LIN {X -0.068,Y -157.540,Z 1544.848,A 0.000,B 0.000,C 90.000,E1 152.615} C_DIS
LIN {X 0.098,Y -161.777,Z 1544.828,A 0.000,B 0.000,C 90.000,E1 148.997} C_DIS
LIN {X -0.019,Y -165.970,Z 1544.808,A 0.000,B 0.000,C 90.000,E1 145.515} C_DIS
LIN {X -0.024,Y -170.964,Z 1544.789,A 0.000,B 0.000,C 90.000,E1 142.029} C_DIS
LIN {X 0.028,Y -175.833,Z 1544.770,A 0.000,B 0.000,C 90.000,E1 138.566} C_DIS
LIN {X 0.023,Y -181.439,Z 1544.751,A 0.000,B 0.000,C 90.000,E1 135.162} C_DIS
LIN {X -0.103,Y -186.945,Z 1544.732,A 0.000,B 0.000,C 90.000,E1 131.838} C_DIS
LIN {X -0.104,Y -190.058,Z 1544.723,A 0.000,B 0.000,C 90.000,E1 130.172} C_DIS
LIN {X -0.090,Y -195.833,Z 1544.705,A 0.000,B 0.000,C 90.000,E1 126.870} C_DIS
LIN {X -0.023,Y -200.665,Z 1544.691,A 0.000,B 0.000,C 90.000,E1 124.405} C_DIS
LIN {X -0.041,Y -203.117,Z 1544.683,A 0.000,B 0.000,C 90.000,E1 123.007} C_DIS
LIN {X 0.168,Y -318.490,Z 1544.683,A 0.000,B 0.000,C 90.000,E1 122.959} C_DIS
LIN {X 0.099,Y -319.542,Z 1544.683,A 0.000,B 0.000,C 90.000,E1 122.959} C_DIS
LIN {X 0.174,Y -324.477,Z 1544.682,A 0.000,B 0.000,C 90.000,E1 122.752} C_DIS
LIN {X -0.044,Y -327.554,Z 1544.681,A 0.000,B 0.000,C 90.000,E1 122.546} C_DIS
LIN {X -0.058,Y -331.261,Z 1544.678,A 0.000,B 0.000,C 90.000,E1 122.084} C_DIS
LIN {X 0.052,Y -333.020,Z 1544.676,A 0.000,B 0.000,C 90.000,E1 121.750} C_DIS
LIN {X 0.134,Y -336.789,Z 1544.671,A 0.000,B 0.000,C 90.000,E1 120.797} C_DIS
LIN {X 0.103,Y -348.404,Z 1544.656,A 0.000,B 0.000,C 90.000,E1 118.025} C_DIS
LIN {X -0.101,Y -361.451,Z 1544.641,A 0.000,B 0.000,C 90.000,E1 115.335} C_DIS
LIN {X 0.095,Y -376.031,Z 1544.626,A 0.000,B 0.000,C 90.000,E1 112.642} C_DIS
LIN {X -0.090,Y -390.387,Z 1544.613,A 0.000,B 0.000,C 90.000,E1 110.355} C_DIS
LIN {X 0.177,Y -406.158,Z 1544.600,A 0.000,B 0.000,C 90.000,E1 108.055} C_DIS
LIN {X 0.216,Y -423.455,Z 1544.588,A 0.000,B 0.000,C 90.000,E1 105.843} C_DIS
LIN {X 0.058,Y -442.382,Z 1544.576,A 0.000,B 0.000,C 90.000,E1 103.716} C_DIS
LIN {X -0.096,Y -462.375,Z 1544.565,A 0.000,B 0.000,C 90.000,E1 101.715} C_DIS
LIN {X 0.079,Y -485.531,Z 1544.553,A 0.000,B 0.000,C 90.000,E1 99.613} C_DIS
LIN {X 0.000,Y -493.167,Z 1544.550,A 0.000,B 0.000,C 90.000,E1 98.973} C_DIS
LIN {X 0.111,Y -494.997,Z 1544.549,A 0.000,B 0.000,C 90.000,E1 98.746} C_DIS
LIN {X 0.025,Y -496.592,Z 1544.547,A 0.000,B 0.000,C 90.000,E1 98.511} C_DIS
LIN {X -0.065,Y -497.782,Z 1544.546,A 0.000,B 0.000,C 90.000,E1 98.276} C_DIS
LIN {X 0.196,Y -499.207,Z 1544.543,A 0.000,B 0.000,C 90.000,E1 97.757} C_DIS
LIN {X -0.028,Y -499.572,Z 1544.541,A 0.000,B 0.000,C 90.000,E1 97.296} C_DIS
LIN {X -0.244,Y -498.940,Z 1544.538,A 0.000,B 0.000,C 90.000,E1 96.834} C_DIS
LIN {X 0.037,Y -497.207,Z 1544.535,A 0.000,B 0.000,C 90.000,E1 96.315} C_DIS
LIN {X -0.097,Y -495.828,Z 1544.534,A 0.000,B 0.000,C 90.000,E1 96.087} C_DIS
LIN {X -0.001,Y -484.503,Z 1544.524,A 0.000,B 0.000,C 90.000,E1 94.359} C_DIS
LIN {X 0.011,Y -475.130,Z 1544.516,A 0.000,B 0.000,C 90.000,E1 92.865} C_DIS
LIN {X 0.033,Y -466.858,Z 1544.509,A 0.000,B 0.000,C 90.000,E1 91.604} C_DIS
LIN {X 0.171,Y -456.481,Z 1544.500,A 0.000,B 0.000,C 90.000,E1 90.057} C_DIS
LIN {X -0.075,Y -447.464,Z 1544.493,A 0.000,B 0.000,C 90.000,E1 88.797} C_DIS
LIN {X 0.005,Y -438.078,Z 1544.486,A 0.000,B 0.000,C 90.000,E1 87.478} C_DIS
LIN {X 0.117,Y -426.571,Z 1544.477,A 0.000,B 0.000,C 90.000,E1 85.869} C_DIS
LIN {X 0.117,Y -413.092,Z 1544.467,A 0.000,B 0.000,C 90.000,E1 83.976} C_DIS
LIN {X 0.005,Y -398.136,Z 1544.454,A 0.000,B 0.000,C 90.000,E1 81.781} C_DIS
LIN {X 0.140,Y -380.438,Z 1544.439,A 0.000,B 0.000,C 90.000,E1 78.926} C_DIS
LIN {X -0.080,Y -363.765,Z 1544.422,A 0.000,B 0.000,C 90.000,E1 76.047} C_DIS
LIN {X 0.113,Y -350.852,Z 1544.409,A 0.000,B 0.000,C 90.000,E1 73.630} C_DIS
LIN {X 0.038,Y -341.231,Z 1544.399,A 0.000,B 0.000,C 90.000,E1 71.819} C_DIS
LIN {X 0.006,Y -325.755,Z 1544.382,A 0.000,B 0.000,C 90.000,E1 68.720} C_DIS
LIN {X -0.096,Y -309.683,Z 1544.362,A 0.000,B 0.000,C 90.000,E1 65.229} C_DIS
LIN {X 0.022,Y -299.787,Z 1544.350,A 0.000,B 0.000,C 90.000,E1 62.922} C_DIS
LIN {X 0.049,Y -288.590,Z 1544.335,A 0.000,B 0.000,C 90.000,E1 60.255} C_DIS
LIN {X -0.083,Y -280.298,Z 1544.323,A 0.000,B 0.000,C 90.000,E1 58.250} C_DIS
LIN {X 0.030,Y -269.427,Z 1544.308,A 0.000,B 0.000,C 90.000,E1 55.468} C_DIS
LIN {X 0.095,Y -258.999,Z 1544.293,A 0.000,B 0.000,C 90.000,E1 52.637} C_DIS
LIN {X -0.168,Y -247.742,Z 1544.275,A 0.000,B 0.000,C 90.000,E1 49.461} C_DIS
LIN {X -0.080,Y -237.298,Z 1544.256,A 0.000,B 0.000,C 90.000,E1 46.134} C_DIS
LIN {X -0.066,Y -228.747,Z 1544.240,A 0.000,B 0.000,C 90.000,E1 43.137} C_DIS
LIN {X -0.059,Y -221.025,Z 1544.223,A 0.000,B 0.000,C 90.000,E1 40.092} C_DIS
LIN {X -0.046,Y -214.000,Z 1544.205,A 0.000,B 0.000,C 90.000,E1 36.996} C_DIS
LIN {X 0.043,Y -207.763,Z 1544.188,A 0.000,B 0.000,C 90.000,E1 33.833} C_DIS
LIN {X -0.017,Y -202.302,Z 1544.170,A 0.000,B 0.000,C 90.000,E1 30.669} C_DIS
LIN {X -0.055,Y -197.586,Z 1544.152,A 0.000,B 0.000,C 90.000,E1 27.462} C_DIS
LIN {X -0.029,Y -192.589,Z 1544.130,A 0.000,B 0.000,C 90.000,E1 23.387} C_DIS
LIN {X -0.010,Y -188.278,Z 1544.107,A 0.000,B 0.000,C 90.000,E1 19.268} C_DIS
LIN {X -0.067,Y -184.100,Z 1544.079,A 0.000,B 0.000,C 90.000,E1 14.300} C_DIS
LIN {X -0.049,Y -180.889,Z 1544.051,A 0.000,B 0.000,C 90.000,E1 9.265} C_DIS
LIN {X 0.079,Y -178.282,Z 1544.014,A 0.000,B 0.000,C 90.000,E1 2.465} C_DIS
LIN {X -0.010,Y -178.518,Z 1543.955,A 0.000,B 0.000,C 90.000,E1 351.894} C_DIS
LIN {X 0.095,Y -180.978,Z 1543.922,A 0.000,B 0.000,C 90.000,E1 345.936} C_DIS
LIN {X 0.017,Y -184.467,Z 1543.894,A 0.000,B 0.000,C 90.000,E1 340.913} C_DIS
LIN {X 0.011,Y -188.390,Z 1543.871,A 0.000,B 0.000,C 90.000,E1 336.741} C_DIS
LIN {X -0.016,Y -193.357,Z 1543.848,A 0.000,B 0.000,C 90.000,E1 332.615} C_DIS
LIN {X -0.043,Y -199.165,Z 1543.825,A 0.000,B 0.000,C 90.000,E1 328.535} C_DIS
LIN {X -0.061,Y -204.509,Z 1543.807,A 0.000,B 0.000,C 90.000,E1 325.308} C_DIS
LIN {X -0.042,Y -210.670,Z 1543.789,A 0.000,B 0.000,C 90.000,E1 322.110} C_DIS
LIN {X 0.060,Y -217.651,Z 1543.772,A 0.000,B 0.000,C 90.000,E1 318.933} C_DIS
LIN {X -0.094,Y -226.415,Z 1543.753,A 0.000,B 0.000,C 90.000,E1 315.486} C_DIS
LIN {X 0.019,Y -236.333,Z 1543.734,A 0.000,B 0.000,C 90.000,E1 312.043} C_DIS
LIN {X 0.035,Y -242.594,Z 1543.723,A 0.000,B 0.000,C 90.000,E1 310.172} C_DIS
LIN {X 0.000,Y -248.230,Z 1543.715,A 0.000,B 0.000,C 90.000,E1 308.705} C_DIS
LIN {X 0.053,Y -256.174,Z 1543.705,A 0.000,B 0.000,C 90.000,E1 306.870} C_DIS
LIN {X -0.071,Y -265.290,Z 1543.695,A 0.000,B 0.000,C 90.000,E1 305.105} C_DIS
LIN {X 0.166,Y -275.499,Z 1543.685,A 0.000,B 0.000,C 90.000,E1 303.293} C_DIS
LIN {X -0.023,Y -291.443,Z 1543.672,A 0.000,B 0.000,C 90.000,E1 300.924} C_DIS
LIN {X 0.132,Y -311.376,Z 1543.657,A 0.000,B 0.000,C 90.000,E1 298.231} C_DIS
LIN {X -0.178,Y -326.813,Z 1543.646,A 0.000,B 0.000,C 90.000,E1 296.360} C_DIS
LIN {X 0.031,Y -345.069,Z 1543.634,A 0.000,B 0.000,C 90.000,E1 294.155} C_DIS
LIN {X 0.097,Y -363.451,Z 1543.623,A 0.000,B 0.000,C 90.000,E1 292.099} C_DIS
LIN {X -0.075,Y -376.354,Z 1543.615,A 0.000,B 0.000,C 90.000,E1 290.737} C_DIS
LIN {X 0.093,Y -386.609,Z 1543.609,A 0.000,B 0.000,C 90.000,E1 289.577} C_DIS
LIN {X 0.042,Y -393.934,Z 1543.604,A 0.000,B 0.000,C 90.000,E1 288.725} C_DIS
LIN {X 0.046,Y -400.651,Z 1543.599,A 0.000,B 0.000,C 90.000,E1 287.873} C_DIS
LIN {X -0.003,Y -406.701,Z 1543.595,A 0.000,B 0.000,C 90.000,E1 287.040} C_DIS
LIN {X 0.000,Y -412.021,Z 1543.590,A 0.000,B 0.000,C 90.000,E1 286.205} C_DIS
LIN {X -0.064,Y -415.120,Z 1543.587,A 0.000,B 0.000,C 90.000,E1 285.662} C_DIS
LIN {X 0.020,Y -419.032,Z 1543.582,A 0.000,B 0.000,C 90.000,E1 284.828} C_DIS
LIN {X 0.032,Y -422.199,Z 1543.578,A 0.000,B 0.000,C 90.000,E1 284.008} C_DIS
LIN {X -0.083,Y -423.934,Z 1543.575,A 0.000,B 0.000,C 90.000,E1 283.480} C_DIS
LIN {X -0.089,Y -425.263,Z 1543.572,A 0.000,B 0.000,C 90.000,E1 282.939} C_DIS
LIN {X 0.233,Y -426.168,Z 1543.569,A 0.000,B 0.000,C 90.000,E1 282.355} C_DIS
LIN {X 0.147,Y -426.651,Z 1543.566,A 0.000,B 0.000,C 90.000,E1 281.827} C_DIS
LIN {X 0.065,Y -426.619,Z 1543.563,A 0.000,B 0.000,C 90.000,E1 281.299} C_DIS
LIN {X -0.095,Y -426.088,Z 1543.560,A 0.000,B 0.000,C 90.000,E1 280.782} C_DIS
LIN {X -0.173,Y -424.963,Z 1543.557,A 0.000,B 0.000,C 90.000,E1 280.254} C_DIS
LIN {X 0.160,Y -423.171,Z 1543.554,A 0.000,B 0.000,C 90.000,E1 279.670} C_DIS
LIN {X -0.001,Y -420.757,Z 1543.551,A 0.000,B 0.000,C 90.000,E1 279.151} C_DIS
LIN {X -0.111,Y -417.535,Z 1543.548,A 0.000,B 0.000,C 90.000,E1 278.624} C_DIS
LIN {X 0.111,Y -413.410,Z 1543.545,A 0.000,B 0.000,C 90.000,E1 278.049} C_DIS
LIN {X -0.094,Y -408.430,Z 1543.542,A 0.000,B 0.000,C 90.000,E1 277.530} C_DIS
LIN {X -0.168,Y -402.630,Z 1543.539,A 0.000,B 0.000,C 90.000,E1 277.004} C_DIS
LIN {X 0.090,Y -396.635,Z 1543.536,A 0.000,B 0.000,C 90.000,E1 276.486} C_DIS
LIN {X -0.193,Y -390.365,Z 1543.534,A 0.000,B 0.000,C 90.000,E1 276.087} C_DIS
LIN {X -0.094,Y -384.023,Z 1543.531,A 0.000,B 0.000,C 90.000,E1 275.682} C_DIS
LIN {X -0.026,Y -374.466,Z 1543.529,A 0.000,B 0.000,C 90.000,E1 275.163} C_DIS
LIN {X 0.057,Y -364.853,Z 1543.526,A 0.000,B 0.000,C 90.000,E1 274.702} C_DIS
LIN {X -0.156,Y -352.144,Z 1543.523,A 0.000,B 0.000,C 90.000,E1 274.188} C_DIS
LIN {X -0.069,Y -342.518,Z 1543.521,A 0.000,B 0.000,C 90.000,E1 273.784} C_DIS
LIN {X 0.158,Y -332.329,Z 1543.519,A 0.000,B 0.000,C 90.000,E1 273.383} C_DIS
LIN {X 0.116,Y -319.217,Z 1543.517,A 0.000,B 0.000,C 90.000,E1 272.980} C_DIS
LIN {X -0.130,Y -309.122,Z 1543.515,A 0.000,B 0.000,C 90.000,E1 272.751} C_DIS
LIN {X 0.095,Y -297.890,Z 1543.514,A 0.000,B 0.000,C 90.000,E1 272.465} C_DIS
LIN {X -0.025,Y -285.540,Z 1543.513,A 0.000,B 0.000,C 90.000,E1 272.293} C_DIS
LIN {X -0.121,Y -272.247,Z 1543.512,A 0.000,B 0.000,C 90.000,E1 272.178} C_DIS
LIN {X 0.101,Y -260.337,Z 1543.512,A 0.000,B 0.000,C 90.000,E1 272.064} C_DIS
LIN {X 0.037,Y -181.250,Z 1543.511,A 0.000,B 0.000,C 90.000,E1 272.064} C_DIS
LIN {X 0.052,Y -181.579,Z 1543.502,A 0.000,B 0.000,C 90.000,E1 270.344} C_DIS
LIN {X 0.027,Y -180.905,Z 1543.474,A 0.000,B 0.000,C 90.000,E1 265.298} C_DIS
LIN {X -0.023,Y -180.248,Z 1543.465,A 0.000,B 0.000,C 90.000,E1 263.628} C_DIS
LIN {X -0.004,Y -178.736,Z 1543.441,A 0.000,B 0.000,C 90.000,E1 259.398} C_DIS
LIN {X 0.063,Y -175.783,Z 1543.413,A 0.000,B 0.000,C 90.000,E1 254.283} C_DIS
LIN {X 0.051,Y -171.968,Z 1543.384,A 0.000,B 0.000,C 90.000,E1 249.156} C_DIS
LIN {X 0.088,Y -171.367,Z 1543.380,A 0.000,B 0.000,C 90.000,E1 248.284} C_DIS
LIN {X -0.085,Y -167.614,Z 1543.355,A 0.000,B 0.000,C 90.000,E1 244.024} C_DIS
LIN {X 0.077,Y -166.264,Z 1543.346,A 0.000,B 0.000,C 90.000,E1 242.231} C_DIS
LIN {X 0.064,Y -163.016,Z 1543.326,A 0.000,B 0.000,C 90.000,E1 238.742} C_DIS
LIN {X -0.023,Y -160.941,Z 1543.312,A 0.000,B 0.000,C 90.000,E1 236.135} C_DIS
LIN {X 0.087,Y -157.699,Z 1543.292,A 0.000,B 0.000,C 90.000,E1 232.557} C_DIS
LIN {X 0.025,Y -155.738,Z 1543.277,A 0.000,B 0.000,C 90.000,E1 229.908} C_DIS
LIN {X 0.078,Y -151.996,Z 1543.252,A 0.000,B 0.000,C 90.000,E1 225.405} C_DIS
LIN {X 0.094,Y -150.241,Z 1543.237,A 0.000,B 0.000,C 90.000,E1 222.690} C_DIS
LIN {X 0.017,Y -147.000,Z 1543.212,A 0.000,B 0.000,C 90.000,E1 218.177} C_DIS
LIN {X 0.006,Y -145.585,Z 1543.197,A 0.000,B 0.000,C 90.000,E1 215.438} C_DIS
LIN {X 0.000,Y -142.973,Z 1543.171,A 0.000,B 0.000,C 90.000,E1 210.846} C_DIS
LIN {X 0.054,Y -141.600,Z 1543.151,A 0.000,B 0.000,C 90.000,E1 207.129} C_DIS
LIN {X -0.031,Y -139.423,Z 1543.115,A 0.000,B 0.000,C 90.000,E1 200.663} C_DIS
LIN {X 0.020,Y -139.151,Z 1543.104,A 0.000,B 0.000,C 90.000,E1 198.779} C_DIS
LIN {X 0.043,Y -138.345,Z 1543.058,A 0.000,B 0.000,C 90.000,E1 190.366} C_DIS
LIN {X 0.028,Y -139.485,Z 1543.006,A 0.000,B 0.000,C 90.000,E1 181.031} C_DIS
LIN {X -0.032,Y -141.084,Z 1542.975,A 0.000,B 0.000,C 90.000,E1 175.469} C_DIS
LIN {X 0.062,Y -142.461,Z 1542.959,A 0.000,B 0.000,C 90.000,E1 172.648} C_DIS
LIN {X 0.011,Y -144.706,Z 1542.934,A 0.000,B 0.000,C 90.000,E1 168.049} C_DIS
LIN {X -0.037,Y -147.303,Z 1542.913,A 0.000,B 0.000,C 90.000,E1 164.393} C_DIS
LIN {X -0.022,Y -150.623,Z 1542.888,A 0.000,B 0.000,C 90.000,E1 159.826} C_DIS
LIN {X 0.055,Y -154.098,Z 1542.868,A 0.000,B 0.000,C 90.000,E1 156.177} C_DIS
LIN {X -0.022,Y -157.521,Z 1542.848,A 0.000,B 0.000,C 90.000,E1 152.615} C_DIS
LIN {X -0.077,Y -161.755,Z 1542.828,A 0.000,B 0.000,C 90.000,E1 149.076} C_DIS
LIN {X 0.029,Y -165.948,Z 1542.808,A 0.000,B 0.000,C 90.000,E1 145.515} C_DIS
LIN {X 0.026,Y -170.939,Z 1542.789,A 0.000,B 0.000,C 90.000,E1 142.029} C_DIS
LIN {X -0.054,Y -175.807,Z 1542.770,A 0.000,B 0.000,C 90.000,E1 138.609} C_DIS
LIN {X 0.074,Y -181.415,Z 1542.751,A 0.000,B 0.000,C 90.000,E1 135.162} C_DIS
LIN {X -0.052,Y -186.918,Z 1542.732,A 0.000,B 0.000,C 90.000,E1 131.838} C_DIS
LIN {X 0.022,Y -191.496,Z 1542.719,A 0.000,B 0.000,C 90.000,E1 129.322} C_DIS
LIN {X 0.106,Y -197.359,Z 1542.700,A 0.000,B 0.000,C 90.000,E1 126.011} C_DIS
LIN {X 0.032,Y -200.636,Z 1542.691,A 0.000,B 0.000,C 90.000,E1 124.405} C_DIS
LIN {X -0.025,Y -203.053,Z 1542.683,A 0.000,B 0.000,C 90.000,E1 123.038} C_DIS
LIN {X -0.077,Y -318.319,Z 1542.683,A 0.000,B 0.000,C 90.000,E1 123.038} C_DIS
LIN {X -0.012,Y -324.630,Z 1542.682,A 0.000,B 0.000,C 90.000,E1 122.801} C_DIS
LIN {X 0.056,Y -327.580,Z 1542.681,A 0.000,B 0.000,C 90.000,E1 122.546} C_DIS
LIN {X -0.033,Y -331.300,Z 1542.678,A 0.000,B 0.000,C 90.000,E1 122.084} C_DIS
LIN {X 0.077,Y -333.015,Z 1542.677,A 0.000,B 0.000,C 90.000,E1 121.750} C_DIS
LIN {X -0.029,Y -339.215,Z 1542.668,A 0.000,B 0.000,C 90.000,E1 120.207} C_DIS
LIN {X 0.003,Y -351.135,Z 1542.652,A 0.000,B 0.000,C 90.000,E1 117.436} C_DIS
LIN {X 0.044,Y -364.510,Z 1542.637,A 0.000,B 0.000,C 90.000,E1 114.719} C_DIS
LIN {X -0.009,Y -379.447,Z 1542.623,A 0.000,B 0.000,C 90.000,E1 112.078} C_DIS
LIN {X 0.114,Y -394.145,Z 1542.610,A 0.000,B 0.000,C 90.000,E1 109.758} C_DIS
LIN {X 0.105,Y -410.284,Z 1542.597,A 0.000,B 0.000,C 90.000,E1 107.511} C_DIS
LIN {X 0.128,Y -427.977,Z 1542.585,A 0.000,B 0.000,C 90.000,E1 105.315} C_DIS
LIN {X 0.237,Y -447.270,Z 1542.573,A 0.000,B 0.000,C 90.000,E1 103.175} C_DIS
LIN {X -0.135,Y -467.405,Z 1542.562,A 0.000,B 0.000,C 90.000,E1 101.243} C_DIS
LIN {X -0.167,Y -490.700,Z 1542.551,A 0.000,B 0.000,C 90.000,E1 99.208} C_DIS
LIN {X 0.018,Y -493.100,Z 1542.550,A 0.000,B 0.000,C 90.000,E1 98.973} C_DIS
LIN {X 0.129,Y -494.921,Z 1542.549,A 0.000,B 0.000,C 90.000,E1 98.746} C_DIS
LIN {X 0.042,Y -496.509,Z 1542.547,A 0.000,B 0.000,C 90.000,E1 98.511} C_DIS
LIN {X -0.047,Y -497.693,Z 1542.546,A 0.000,B 0.000,C 90.000,E1 98.276} C_DIS
LIN {X 0.214,Y -499.108,Z 1542.543,A 0.000,B 0.000,C 90.000,E1 97.757} C_DIS
LIN {X -0.011,Y -499.466,Z 1542.541,A 0.000,B 0.000,C 90.000,E1 97.296} C_DIS
LIN {X -0.228,Y -498.826,Z 1542.538,A 0.000,B 0.000,C 90.000,E1 96.834} C_DIS
LIN {X 0.053,Y -497.084,Z 1542.535,A 0.000,B 0.000,C 90.000,E1 96.315} C_DIS
LIN {X -0.083,Y -495.699,Z 1542.534,A 0.000,B 0.000,C 90.000,E1 96.087} C_DIS
LIN {X 0.011,Y -484.387,Z 1542.524,A 0.000,B 0.000,C 90.000,E1 94.359} C_DIS
LIN {X 0.021,Y -475.033,Z 1542.516,A 0.000,B 0.000,C 90.000,E1 92.865} C_DIS
LIN {X 0.042,Y -466.753,Z 1542.509,A 0.000,B 0.000,C 90.000,E1 91.604} C_DIS
LIN {X -0.060,Y -458.152,Z 1542.502,A 0.000,B 0.000,C 90.000,E1 90.344} C_DIS
LIN {X 0.167,Y -449.206,Z 1542.495,A 0.000,B 0.000,C 90.000,E1 89.026} C_DIS
LIN {X 0.009,Y -438.010,Z 1542.486,A 0.000,B 0.000,C 90.000,E1 87.478} C_DIS
LIN {X -0.044,Y -428.469,Z 1542.479,A 0.000,B 0.000,C 90.000,E1 86.159} C_DIS
LIN {X 0.118,Y -413.097,Z 1542.467,A 0.000,B 0.000,C 90.000,E1 83.976} C_DIS
LIN {X 0.007,Y -398.158,Z 1542.454,A 0.000,B 0.000,C 90.000,E1 81.781} C_DIS
LIN {X 0.169,Y -378.752,Z 1542.437,A 0.000,B 0.000,C 90.000,E1 78.634} C_DIS
LIN {X -0.128,Y -360.518,Z 1542.419,A 0.000,B 0.000,C 90.000,E1 75.463} C_DIS
LIN {X 0.074,Y -347.664,Z 1542.406,A 0.000,B 0.000,C 90.000,E1 73.032} C_DIS
LIN {X -0.062,Y -334.921,Z 1542.392,A 0.000,B 0.000,C 90.000,E1 70.604} C_DIS
LIN {X -0.068,Y -322.732,Z 1542.378,A 0.000,B 0.000,C 90.000,E1 68.103} C_DIS
LIN {X -0.046,Y -308.288,Z 1542.360,A 0.000,B 0.000,C 90.000,E1 64.897} C_DIS
LIN {X 0.026,Y -299.816,Z 1542.350,A 0.000,B 0.000,C 90.000,E1 62.922} C_DIS
LIN {X 0.053,Y -288.621,Z 1542.335,A 0.000,B 0.000,C 90.000,E1 60.255} C_DIS
LIN {X -0.078,Y -280.353,Z 1542.323,A 0.000,B 0.000,C 90.000,E1 58.250} C_DIS
LIN {X 0.034,Y -269.479,Z 1542.308,A 0.000,B 0.000,C 90.000,E1 55.468} C_DIS
LIN {X 0.101,Y -259.061,Z 1542.293,A 0.000,B 0.000,C 90.000,E1 52.637} C_DIS
LIN {X -0.159,Y -247.852,Z 1542.275,A 0.000,B 0.000,C 90.000,E1 49.461} C_DIS
LIN {X -0.069,Y -237.441,Z 1542.256,A 0.000,B 0.000,C 90.000,E1 46.134} C_DIS
LIN {X -0.052,Y -228.915,Z 1542.240,A 0.000,B 0.000,C 90.000,E1 43.137} C_DIS
LIN {X -0.041,Y -221.238,Z 1542.223,A 0.000,B 0.000,C 90.000,E1 40.092} C_DIS
LIN {X -0.024,Y -214.234,Z 1542.205,A 0.000,B 0.000,C 90.000,E1 36.996} C_DIS
LIN {X -0.045,Y -208.020,Z 1542.188,A 0.000,B 0.000,C 90.000,E1 33.865} C_DIS
LIN {X 0.018,Y -202.591,Z 1542.170,A 0.000,B 0.000,C 90.000,E1 30.669} C_DIS
LIN {X -0.064,Y -196.814,Z 1542.148,A 0.000,B 0.000,C 90.000,E1 26.668} C_DIS
LIN {X -0.052,Y -191.951,Z 1542.125,A 0.000,B 0.000,C 90.000,E1 22.589} C_DIS
LIN {X -0.053,Y -187.793,Z 1542.103,A 0.000,B 0.000,C 90.000,E1 18.471} C_DIS
LIN {X -0.008,Y -183.771,Z 1542.075,A 0.000,B 0.000,C 90.000,E1 13.467} C_DIS
LIN {X -0.077,Y -180.723,Z 1542.047,A 0.000,B 0.000,C 90.000,E1 8.454} C_DIS
LIN {X 0.063,Y -178.225,Z 1542.005,A 0.000,B 0.000,C 90.000,E1 0.802} C_DIS
LIN {X 0.065,Y -179.013,Z 1541.950,A 0.000,B 0.000,C 90.000,E1 351.027} C_DIS
LIN {X 0.045,Y -181.724,Z 1541.917,A 0.000,B 0.000,C 90.000,E1 345.117} C_DIS
LIN {X 0.102,Y -185.411,Z 1541.889,A 0.000,B 0.000,C 90.000,E1 340.061} C_DIS
LIN {X 0.023,Y -189.514,Z 1541.866,A 0.000,B 0.000,C 90.000,E1 335.921} C_DIS
LIN {X -0.051,Y -194.625,Z 1541.843,A 0.000,B 0.000,C 90.000,E1 331.820} C_DIS
LIN {X -0.036,Y -200.605,Z 1541.821,A 0.000,B 0.000,C 90.000,E1 327.740} C_DIS
LIN {X 0.094,Y -206.094,Z 1541.803,A 0.000,B 0.000,C 90.000,E1 324.482} C_DIS
LIN {X -0.017,Y -212.439,Z 1541.785,A 0.000,B 0.000,C 90.000,E1 321.331} C_DIS
LIN {X 0.103,Y -219.629,Z 1541.768,A 0.000,B 0.000,C 90.000,E1 318.162} C_DIS
LIN {X 0.077,Y -227.525,Z 1541.751,A 0.000,B 0.000,C 90.000,E1 315.081} C_DIS
LIN {X 0.073,Y -237.534,Z 1541.732,A 0.000,B 0.000,C 90.000,E1 311.676} C_DIS
LIN {X -0.078,Y -243.950,Z 1541.721,A 0.000,B 0.000,C 90.000,E1 309.850} C_DIS
LIN {X -0.103,Y -249.730,Z 1541.713,A 0.000,B 0.000,C 90.000,E1 308.382} C_DIS
LIN {X 0.149,Y -256.136,Z 1541.705,A 0.000,B 0.000,C 90.000,E1 306.870} C_DIS
LIN {X 0.027,Y -265.189,Z 1541.695,A 0.000,B 0.000,C 90.000,E1 305.105} C_DIS
LIN {X -0.115,Y -275.352,Z 1541.685,A 0.000,B 0.000,C 90.000,E1 303.372} C_DIS
LIN {X 0.105,Y -288.912,Z 1541.674,A 0.000,B 0.000,C 90.000,E1 301.258} C_DIS
LIN {X -0.110,Y -303.577,Z 1541.663,A 0.000,B 0.000,C 90.000,E1 299.283} C_DIS
LIN {X -0.132,Y -321.518,Z 1541.650,A 0.000,B 0.000,C 90.000,E1 297.001} C_DIS
LIN {X -0.104,Y -339.561,Z 1541.638,A 0.000,B 0.000,C 90.000,E1 294.823} C_DIS
LIN {X -0.052,Y -360.538,Z 1541.625,A 0.000,B 0.000,C 90.000,E1 292.461} C_DIS
LIN {X -0.186,Y -373.367,Z 1541.617,A 0.000,B 0.000,C 90.000,E1 291.099} C_DIS
LIN {X 0.095,Y -383.627,Z 1541.611,A 0.000,B 0.000,C 90.000,E1 289.939} C_DIS
LIN {X 0.062,Y -391.137,Z 1541.606,A 0.000,B 0.000,C 90.000,E1 289.087} C_DIS
LIN {X 0.049,Y -398.123,Z 1541.601,A 0.000,B 0.000,C 90.000,E1 288.236} C_DIS
LIN {X -0.030,Y -404.469,Z 1541.597,A 0.000,B 0.000,C 90.000,E1 287.402} C_DIS
LIN {X -0.137,Y -408.349,Z 1541.594,A 0.000,B 0.000,C 90.000,E1 286.858} C_DIS
LIN {X -0.116,Y -413.472,Z 1541.589,A 0.000,B 0.000,C 90.000,E1 286.024} C_DIS
LIN {X -0.051,Y -417.787,Z 1541.584,A 0.000,B 0.000,C 90.000,E1 285.190} C_DIS
LIN {X 0.058,Y -421.286,Z 1541.580,A 0.000,B 0.000,C 90.000,E1 284.356} C_DIS
LIN {X 0.093,Y -424.082,Z 1541.575,A 0.000,B 0.000,C 90.000,E1 283.536} C_DIS
LIN {X -0.008,Y -425.497,Z 1541.572,A 0.000,B 0.000,C 90.000,E1 283.008} C_DIS
LIN {X -0.099,Y -426.512,Z 1541.569,A 0.000,B 0.000,C 90.000,E1 282.479} C_DIS
LIN {X -0.182,Y -427.102,Z 1541.566,A 0.000,B 0.000,C 90.000,E1 281.951} C_DIS
LIN {X 0.160,Y -427.157,Z 1541.563,A 0.000,B 0.000,C 90.000,E1 281.366} C_DIS
LIN {X 0.084,Y -426.706,Z 1541.560,A 0.000,B 0.000,C 90.000,E1 280.838} C_DIS
LIN {X 0.009,Y -425.724,Z 1541.557,A 0.000,B 0.000,C 90.000,E1 280.310} C_DIS
LIN {X -0.145,Y -424.083,Z 1541.554,A 0.000,B 0.000,C 90.000,E1 279.792} C_DIS
LIN {X 0.186,Y -421.765,Z 1541.551,A 0.000,B 0.000,C 90.000,E1 279.208} C_DIS
LIN {X 0.080,Y -418.705,Z 1541.548,A 0.000,B 0.000,C 90.000,E1 278.681} C_DIS
LIN {X -0.105,Y -414.791,Z 1541.545,A 0.000,B 0.000,C 90.000,E1 278.163} C_DIS
LIN {X 0.104,Y -409.906,Z 1541.542,A 0.000,B 0.000,C 90.000,E1 277.587} C_DIS
LIN {X -0.064,Y -404.254,Z 1541.539,A 0.000,B 0.000,C 90.000,E1 277.068} C_DIS
LIN {X 0.123,Y -398.204,Z 1541.536,A 0.000,B 0.000,C 90.000,E1 276.549} C_DIS
LIN {X -0.135,Y -392.084,Z 1541.534,A 0.000,B 0.000,C 90.000,E1 276.144} C_DIS
LIN {X -0.184,Y -382.454,Z 1541.531,A 0.000,B 0.000,C 90.000,E1 275.568} C_DIS
LIN {X -0.031,Y -372.665,Z 1541.528,A 0.000,B 0.000,C 90.000,E1 275.049} C_DIS
LIN {X -0.019,Y -359.924,Z 1541.525,A 0.000,B 0.000,C 90.000,E1 274.473} C_DIS
LIN {X -0.059,Y -347.459,Z 1541.522,A 0.000,B 0.000,C 90.000,E1 273.955} C_DIS
LIN {X 0.151,Y -337.822,Z 1541.520,A 0.000,B 0.000,C 90.000,E1 273.555} C_DIS
LIN {X -0.069,Y -324.518,Z 1541.517,A 0.000,B 0.000,C 90.000,E1 273.154} C_DIS
LIN {X -0.101,Y -314.293,Z 1541.516,A 0.000,B 0.000,C 90.000,E1 272.865} C_DIS
LIN {X 0.075,Y -303.757,Z 1541.514,A 0.000,B 0.000,C 90.000,E1 272.579} C_DIS
LIN {X 0.116,Y -291.904,Z 1541.513,A 0.000,B 0.000,C 90.000,E1 272.350} C_DIS
LIN {X 0.101,Y -278.448,Z 1541.512,A 0.000,B 0.000,C 90.000,E1 272.178} C_DIS
LIN {X -0.130,Y -261.589,Z 1541.512,A 0.000,B 0.000,C 90.000,E1 272.121} C_DIS
LIN {X 0.058,Y -181.249,Z 1541.512,A 0.000,B 0.000,C 90.000,E1 272.064} C_DIS
LIN {X -0.078,Y -181.578,Z 1541.502,A 0.000,B 0.000,C 90.000,E1 270.401} C_DIS
LIN {X 0.079,Y -180.905,Z 1541.474,A 0.000,B 0.000,C 90.000,E1 265.298} C_DIS
LIN {X 0.029,Y -180.255,Z 1541.465,A 0.000,B 0.000,C 90.000,E1 263.628} C_DIS
LIN {X 0.048,Y -178.746,Z 1541.441,A 0.000,B 0.000,C 90.000,E1 259.398} C_DIS
LIN {X -0.055,Y -175.793,Z 1541.413,A 0.000,B 0.000,C 90.000,E1 254.338} C_DIS
LIN {X -0.060,Y -171.978,Z 1541.384,A 0.000,B 0.000,C 90.000,E1 249.209} C_DIS
LIN {X -0.022,Y -171.381,Z 1541.380,A 0.000,B 0.000,C 90.000,E1 248.337} C_DIS
LIN {X -0.037,Y -167.627,Z 1541.356,A 0.000,B 0.000,C 90.000,E1 244.024} C_DIS
LIN {X -0.022,Y -166.281,Z 1541.346,A 0.000,B 0.000,C 90.000,E1 242.281} C_DIS
LIN {X -0.027,Y -163.030,Z 1541.327,A 0.000,B 0.000,C 90.000,E1 238.791} C_DIS
LIN {X 0.025,Y -160.958,Z 1541.312,A 0.000,B 0.000,C 90.000,E1 236.135} C_DIS
LIN {X 0.009,Y -157.713,Z 1541.292,A 0.000,B 0.000,C 90.000,E1 232.603} C_DIS
LIN {X 0.072,Y -155.752,Z 1541.277,A 0.000,B 0.000,C 90.000,E1 229.908} C_DIS
LIN {X 0.018,Y -152.009,Z 1541.253,A 0.000,B 0.000,C 90.000,E1 225.445} C_DIS
LIN {X -0.072,Y -150.256,Z 1541.237,A 0.000,B 0.000,C 90.000,E1 222.771} C_DIS
LIN {X 0.062,Y -147.010,Z 1541.212,A 0.000,B 0.000,C 90.000,E1 218.177} C_DIS
LIN {X 0.052,Y -145.594,Z 1541.197,A 0.000,B 0.000,C 90.000,E1 215.438} C_DIS
LIN {X -0.028,Y -142.981,Z 1541.172,A 0.000,B 0.000,C 90.000,E1 210.875} C_DIS
LIN {X -0.028,Y -141.608,Z 1541.151,A 0.000,B 0.000,C 90.000,E1 207.180} C_DIS
LIN {X 0.014,Y -139.426,Z 1541.115,A 0.000,B 0.000,C 90.000,E1 200.663} C_DIS
LIN {X 0.064,Y -139.155,Z 1541.104,A 0.000,B 0.000,C 90.000,E1 198.779} C_DIS
LIN {X -0.050,Y -138.344,Z 1541.058,A 0.000,B 0.000,C 90.000,E1 190.423} C_DIS
LIN {X -0.068,Y -139.483,Z 1541.006,A 0.000,B 0.000,C 90.000,E1 181.088} C_DIS
LIN {X 0.013,Y -141.077,Z 1540.975,A 0.000,B 0.000,C 90.000,E1 175.469} C_DIS
LIN {X -0.034,Y -142.453,Z 1540.959,A 0.000,B 0.000,C 90.000,E1 172.704} C_DIS
LIN {X 0.056,Y -144.694,Z 1540.934,A 0.000,B 0.000,C 90.000,E1 168.049} C_DIS
LIN {X 0.008,Y -147.289,Z 1540.913,A 0.000,B 0.000,C 90.000,E1 164.393} C_DIS
LIN {X 0.025,Y -150.608,Z 1540.888,A 0.000,B 0.000,C 90.000,E1 159.826} C_DIS
LIN {X -0.040,Y -154.082,Z 1540.868,A 0.000,B 0.000,C 90.000,E1 156.230} C_DIS
LIN {X 0.026,Y -157.503,Z 1540.848,A 0.000,B 0.000,C 90.000,E1 152.615} C_DIS
LIN {X -0.028,Y -161.733,Z 1540.828,A 0.000,B 0.000,C 90.000,E1 149.076} C_DIS
LIN {X -0.016,Y -165.926,Z 1540.809,A 0.000,B 0.000,C 90.000,E1 145.548} C_DIS
LIN {X -0.029,Y -170.914,Z 1540.789,A 0.000,B 0.000,C 90.000,E1 142.065} C_DIS
LIN {X -0.003,Y -175.782,Z 1540.770,A 0.000,B 0.000,C 90.000,E1 138.609} C_DIS
LIN {X -0.002,Y -181.391,Z 1540.751,A 0.000,B 0.000,C 90.000,E1 135.202} C_DIS
LIN {X 0.001,Y -186.888,Z 1540.732,A 0.000,B 0.000,C 90.000,E1 131.838} C_DIS
LIN {X -0.046,Y -191.471,Z 1540.719,A 0.000,B 0.000,C 90.000,E1 129.358} C_DIS
LIN {X -0.115,Y -197.328,Z 1540.700,A 0.000,B 0.000,C 90.000,E1 126.091} C_DIS
LIN {X 0.087,Y -200.605,Z 1540.691,A 0.000,B 0.000,C 90.000,E1 124.405} C_DIS
LIN {X -0.063,Y -202.986,Z 1540.684,A 0.000,B 0.000,C 90.000,E1 123.086} C_DIS
LIN {X -0.140,Y -318.104,Z 1540.684,A 0.000,B 0.000,C 90.000,E1 123.086} C_DIS
LIN {X -0.121,Y -322.661,Z 1540.683,A 0.000,B 0.000,C 90.000,E1 122.959} C_DIS
LIN {X -0.099,Y -324.774,Z 1540.682,A 0.000,B 0.000,C 90.000,E1 122.832} C_DIS
LIN {X -0.043,Y -328.644,Z 1540.680,A 0.000,B 0.000,C 90.000,E1 122.467} C_DIS
LIN {X 0.075,Y -332.149,Z 1540.677,A 0.000,B 0.000,C 90.000,E1 121.926} C_DIS
LIN {X 0.187,Y -333.640,Z 1540.676,A 0.000,B 0.000,C 90.000,E1 121.592} C_DIS
LIN {X -0.085,Y -346.233,Z 1540.658,A 0.000,B 0.000,C 90.000,E1 118.537} C_DIS
LIN {X -0.036,Y -359.021,Z 1540.643,A 0.000,B 0.000,C 90.000,E1 115.796} C_DIS
LIN {X -0.094,Y -373.323,Z 1540.628,A 0.000,B 0.000,C 90.000,E1 113.131} C_DIS
LIN {X 0.007,Y -387.414,Z 1540.615,A 0.000,B 0.000,C 90.000,E1 110.791} C_DIS
LIN {X -0.175,Y -402.898,Z 1540.603,A 0.000,B 0.000,C 90.000,E1 108.544} C_DIS
LIN {X -0.107,Y -419.886,Z 1540.591,A 0.000,B 0.000,C 90.000,E1 106.315} C_DIS
LIN {X 0.149,Y -438.495,Z 1540.578,A 0.000,B 0.000,C 90.000,E1 104.120} C_DIS
LIN {X 0.178,Y -458.358,Z 1540.567,A 0.000,B 0.000,C 90.000,E1 102.063} C_DIS
LIN {X -0.008,Y -478.796,Z 1540.557,A 0.000,B 0.000,C 90.000,E1 100.197} C_DIS
LIN {X -0.019,Y -491.819,Z 1540.551,A 0.000,B 0.000,C 90.000,E1 99.095} C_DIS
LIN {X 0.143,Y -493.948,Z 1540.549,A 0.000,B 0.000,C 90.000,E1 98.859} C_DIS
LIN {X -0.183,Y -495.568,Z 1540.548,A 0.000,B 0.000,C 90.000,E1 98.681} C_DIS
LIN {X 0.147,Y -496.966,Z 1540.547,A 0.000,B 0.000,C 90.000,E1 98.398} C_DIS
LIN {X 0.061,Y -497.998,Z 1540.545,A 0.000,B 0.000,C 90.000,E1 98.163} C_DIS
LIN {X -0.168,Y -499.168,Z 1540.543,A 0.000,B 0.000,C 90.000,E1 97.701} C_DIS
LIN {X 0.105,Y -499.308,Z 1540.540,A 0.000,B 0.000,C 90.000,E1 97.182} C_DIS
LIN {X -0.111,Y -498.443,Z 1540.537,A 0.000,B 0.000,C 90.000,E1 96.720} C_DIS
LIN {X 0.169,Y -496.426,Z 1540.535,A 0.000,B 0.000,C 90.000,E1 96.201} C_DIS
LIN {X -0.040,Y -477.430,Z 1540.518,A 0.000,B 0.000,C 90.000,E1 93.269} C_DIS
LIN {X 0.024,Y -469.336,Z 1540.511,A 0.000,B 0.000,C 90.000,E1 92.007} C_DIS
LIN {X 0.217,Y -459.075,Z 1540.503,A 0.000,B 0.000,C 90.000,E1 90.458} C_DIS
LIN {X 0.008,Y -450.172,Z 1540.496,A 0.000,B 0.000,C 90.000,E1 89.198} C_DIS
LIN {X -0.130,Y -439.041,Z 1540.487,A 0.000,B 0.000,C 90.000,E1 87.650} C_DIS
LIN {X -0.025,Y -427.626,Z 1540.478,A 0.000,B 0.000,C 90.000,E1 86.045} C_DIS
LIN {X 0.028,Y -414.198,Z 1540.468,A 0.000,B 0.000,C 90.000,E1 84.147} C_DIS
LIN {X -0.050,Y -399.255,Z 1540.455,A 0.000,B 0.000,C 90.000,E1 81.951} C_DIS
LIN {X 0.090,Y -379.769,Z 1540.438,A 0.000,B 0.000,C 90.000,E1 78.814} C_DIS
LIN {X -0.182,Y -361.453,Z 1540.420,A 0.000,B 0.000,C 90.000,E1 75.644} C_DIS
LIN {X 0.143,Y -348.583,Z 1540.407,A 0.000,B 0.000,C 90.000,E1 73.196} C_DIS
LIN {X -0.072,Y -335.860,Z 1540.393,A 0.000,B 0.000,C 90.000,E1 70.786} C_DIS
LIN {X -0.093,Y -322.142,Z 1540.378,A 0.000,B 0.000,C 90.000,E1 67.975} C_DIS
LIN {X 0.194,Y -307.715,Z 1540.360,A 0.000,B 0.000,C 90.000,E1 64.717} C_DIS
LIN {X -0.023,Y -299.234,Z 1540.349,A 0.000,B 0.000,C 90.000,E1 62.794} C_DIS
LIN {X -0.008,Y -288.062,Z 1540.334,A 0.000,B 0.000,C 90.000,E1 60.127} C_DIS
LIN {X 0.046,Y -278.456,Z 1540.321,A 0.000,B 0.000,C 90.000,E1 57.740} C_DIS
LIN {X 0.027,Y -267.675,Z 1540.305,A 0.000,B 0.000,C 90.000,E1 54.975} C_DIS
LIN {X -0.110,Y -256.064,Z 1540.288,A 0.000,B 0.000,C 90.000,E1 51.823} C_DIS
LIN {X 0.069,Y -245.091,Z 1540.270,A 0.000,B 0.000,C 90.000,E1 48.528} C_DIS
LIN {X -0.094,Y -234.932,Z 1540.251,A 0.000,B 0.000,C 90.000,E1 45.243} C_DIS
LIN {X 0.034,Y -226.684,Z 1540.234,A 0.000,B 0.000,C 90.000,E1 42.204} C_DIS
LIN {X 0.015,Y -219.271,Z 1540.218,A 0.000,B 0.000,C 90.000,E1 39.152} C_DIS
LIN {X -0.143,Y -212.547,Z 1540.200,A 0.000,B 0.000,C 90.000,E1 36.091} C_DIS
LIN {X 0.087,Y -206.568,Z 1540.183,A 0.000,B 0.000,C 90.000,E1 32.880} C_DIS
LIN {X -0.104,Y -201.393,Z 1540.165,A 0.000,B 0.000,C 90.000,E1 29.745} C_DIS
LIN {X 0.041,Y -195.854,Z 1540.143,A 0.000,B 0.000,C 90.000,E1 25.668} C_DIS
LIN {X 0.025,Y -191.143,Z 1540.120,A 0.000,B 0.000,C 90.000,E1 21.589} C_DIS
LIN {X 0.047,Y -187.175,Z 1540.097,A 0.000,B 0.000,C 90.000,E1 17.457} C_DIS
LIN {X -0.018,Y -183.344,Z 1540.069,A 0.000,B 0.000,C 90.000,E1 12.479} C_DIS
LIN {X -0.044,Y -180.136,Z 1540.037,A 0.000,B 0.000,C 90.000,E1 6.606} C_DIS
LIN {X 0.075,Y -178.259,Z 1539.983,A 0.000,B 0.000,C 90.000,E1 356.963} C_DIS
LIN {X -0.021,Y -180.230,Z 1539.936,A 0.000,B 0.000,C 90.000,E1 348.522} C_DIS
LIN {X 0.026,Y -183.064,Z 1539.908,A 0.000,B 0.000,C 90.000,E1 343.449} C_DIS
LIN {X 0.021,Y -186.393,Z 1539.885,A 0.000,B 0.000,C 90.000,E1 339.263} C_DIS
LIN {X 0.045,Y -190.676,Z 1539.862,A 0.000,B 0.000,C 90.000,E1 335.101} C_DIS
LIN {X 0.002,Y -195.927,Z 1539.839,A 0.000,B 0.000,C 90.000,E1 331.001} C_DIS
LIN {X 0.088,Y -202.083,Z 1539.816,A 0.000,B 0.000,C 90.000,E1 326.914} C_DIS
LIN {X 0.091,Y -207.730,Z 1539.798,A 0.000,B 0.000,C 90.000,E1 323.703} C_DIS
LIN {X -0.014,Y -214.273,Z 1539.781,A 0.000,B 0.000,C 90.000,E1 320.561} C_DIS
LIN {X -0.004,Y -221.612,Z 1539.764,A 0.000,B 0.000,C 90.000,E1 317.433} C_DIS
LIN {X 0.027,Y -229.719,Z 1539.746,A 0.000,B 0.000,C 90.000,E1 314.352} C_DIS
LIN {X -0.051,Y -238.771,Z 1539.730,A 0.000,B 0.000,C 90.000,E1 311.353} C_DIS
LIN {X 0.004,Y -245.339,Z 1539.719,A 0.000,B 0.000,C 90.000,E1 309.483} C_DIS
LIN {X 0.008,Y -252.813,Z 1539.709,A 0.000,B 0.000,C 90.000,E1 307.649} C_DIS
LIN {X -0.058,Y -259.570,Z 1539.701,A 0.000,B 0.000,C 90.000,E1 306.217} C_DIS
LIN {X 0.023,Y -267.028,Z 1539.693,A 0.000,B 0.000,C 90.000,E1 304.771} C_DIS
LIN {X -0.082,Y -277.338,Z 1539.683,A 0.000,B 0.000,C 90.000,E1 303.038} C_DIS
LIN {X 0.146,Y -295.875,Z 1539.668,A 0.000,B 0.000,C 90.000,E1 300.256} C_DIS
LIN {X -0.046,Y -313.541,Z 1539.655,A 0.000,B 0.000,C 90.000,E1 297.975} C_DIS
LIN {X -0.072,Y -329.160,Z 1539.645,A 0.000,B 0.000,C 90.000,E1 296.052} C_DIS
LIN {X -0.125,Y -347.285,Z 1539.633,A 0.000,B 0.000,C 90.000,E1 293.951} C_DIS
LIN {X 0.090,Y -362.900,Z 1539.623,A 0.000,B 0.000,C 90.000,E1 292.206} C_DIS
LIN {X 0.149,Y -375.978,Z 1539.616,A 0.000,B 0.000,C 90.000,E1 290.791} C_DIS
LIN {X 0.004,Y -386.244,Z 1539.609,A 0.000,B 0.000,C 90.000,E1 289.685} C_DIS
LIN {X -0.105,Y -393.602,Z 1539.605,A 0.000,B 0.000,C 90.000,E1 288.852} C_DIS
LIN {X -0.103,Y -400.378,Z 1539.600,A 0.000,B 0.000,C 90.000,E1 288.000} C_DIS
LIN {X -0.036,Y -406.558,Z 1539.595,A 0.000,B 0.000,C 90.000,E1 287.149} C_DIS
LIN {X -0.039,Y -411.998,Z 1539.591,A 0.000,B 0.000,C 90.000,E1 286.315} C_DIS
LIN {X 0.016,Y -416.633,Z 1539.586,A 0.000,B 0.000,C 90.000,E1 285.481} C_DIS
LIN {X 0.003,Y -420.464,Z 1539.581,A 0.000,B 0.000,C 90.000,E1 284.662} C_DIS
LIN {X -0.014,Y -422.631,Z 1539.578,A 0.000,B 0.000,C 90.000,E1 284.120} C_DIS
LIN {X -0.123,Y -424.430,Z 1539.575,A 0.000,B 0.000,C 90.000,E1 283.592} C_DIS
LIN {X -0.224,Y -425.863,Z 1539.572,A 0.000,B 0.000,C 90.000,E1 283.063} C_DIS
LIN {X 0.102,Y -426.944,Z 1539.569,A 0.000,B 0.000,C 90.000,E1 282.479} C_DIS
LIN {X 0.023,Y -427.542,Z 1539.566,A 0.000,B 0.000,C 90.000,E1 281.951} C_DIS
LIN {X -0.053,Y -427.657,Z 1539.563,A 0.000,B 0.000,C 90.000,E1 281.422} C_DIS
LIN {X -0.126,Y -427.277,Z 1539.560,A 0.000,B 0.000,C 90.000,E1 280.894} C_DIS
LIN {X 0.220,Y -426.330,Z 1539.557,A 0.000,B 0.000,C 90.000,E1 280.310} C_DIS
LIN {X 0.069,Y -424.786,Z 1539.554,A 0.000,B 0.000,C 90.000,E1 279.792} C_DIS
LIN {X -0.015,Y -422.530,Z 1539.552,A 0.000,B 0.000,C 90.000,E1 279.265} C_DIS
LIN {X -0.179,Y -419.532,Z 1539.548,A 0.000,B 0.000,C 90.000,E1 278.746} C_DIS
LIN {X 0.118,Y -415.727,Z 1539.545,A 0.000,B 0.000,C 90.000,E1 278.163} C_DIS
LIN {X -0.078,Y -410.922,Z 1539.542,A 0.000,B 0.000,C 90.000,E1 277.644} C_DIS
LIN {X 0.111,Y -405.195,Z 1539.539,A 0.000,B 0.000,C 90.000,E1 277.068} C_DIS
LIN {X -0.091,Y -399.254,Z 1539.537,A 0.000,B 0.000,C 90.000,E1 276.606} C_DIS
LIN {X 0.007,Y -393.062,Z 1539.534,A 0.000,B 0.000,C 90.000,E1 276.144} C_DIS
LIN {X -0.017,Y -386.561,Z 1539.532,A 0.000,B 0.000,C 90.000,E1 275.739} C_DIS
LIN {X -0.047,Y -376.786,Z 1539.529,A 0.000,B 0.000,C 90.000,E1 275.220} C_DIS
LIN {X -0.141,Y -363.998,Z 1539.526,A 0.000,B 0.000,C 90.000,E1 274.645} C_DIS
LIN {X 0.001,Y -348.220,Z 1539.522,A 0.000,B 0.000,C 90.000,E1 273.955} C_DIS
LIN {X -0.168,Y -338.448,Z 1539.520,A 0.000,B 0.000,C 90.000,E1 273.612} C_DIS
LIN {X -0.042,Y -325.182,Z 1539.517,A 0.000,B 0.000,C 90.000,E1 273.154} C_DIS
LIN {X -0.078,Y -315.033,Z 1539.516,A 0.000,B 0.000,C 90.000,E1 272.865} C_DIS
LIN {X 0.089,Y -304.437,Z 1539.514,A 0.000,B 0.000,C 90.000,E1 272.579} C_DIS
LIN {X 0.138,Y -292.656,Z 1539.513,A 0.000,B 0.000,C 90.000,E1 272.350} C_DIS
LIN {X 0.125,Y -279.333,Z 1539.512,A 0.000,B 0.000,C 90.000,E1 272.178} C_DIS
LIN {X -0.058,Y -265.096,Z 1539.512,A 0.000,B 0.000,C 90.000,E1 272.121} C_DIS
LIN {X 0.108,Y -258.653,Z 1539.512,A 0.000,B 0.000,C 90.000,E1 272.064} C_DIS
LIN {X 0.043,Y -181.249,Z 1539.512,A 0.000,B 0.000,C 90.000,E1 272.064} C_DIS
LIN {X -0.033,Y -181.567,Z 1539.500,A 0.000,B 0.000,C 90.000,E1 270.057} C_DIS
LIN {X -0.045,Y -180.860,Z 1539.472,A 0.000,B 0.000,C 90.000,E1 265.008} C_DIS
LIN {X 0.008,Y -178.973,Z 1539.444,A 0.000,B 0.000,C 90.000,E1 259.926} C_DIS
LIN {X 0.019,Y -177.934,Z 1539.435,A 0.000,B 0.000,C 90.000,E1 258.229} C_DIS
LIN {X 0.034,Y -175.572,Z 1539.411,A 0.000,B 0.000,C 90.000,E1 253.976} C_DIS
LIN {X 0.040,Y -172.300,Z 1539.387,A 0.000,B 0.000,C 90.000,E1 249.699} C_DIS
LIN {X 0.017,Y -171.779,Z 1539.383,A 0.000,B 0.000,C 90.000,E1 248.847} C_DIS
LIN {X -0.010,Y -168.709,Z 1539.363,A 0.000,B 0.000,C 90.000,E1 245.409} C_DIS
LIN {X 0.028,Y -166.773,Z 1539.349,A 0.000,B 0.000,C 90.000,E1 242.794} C_DIS
LIN {X -0.052,Y -162.753,Z 1539.325,A 0.000,B 0.000,C 90.000,E1 238.456} C_DIS
LIN {X -0.075,Y -161.443,Z 1539.315,A 0.000,B 0.000,C 90.000,E1 236.707} C_DIS
LIN {X -0.034,Y -157.437,Z 1539.290,A 0.000,B 0.000,C 90.000,E1 232.271} C_DIS
LIN {X 0.001,Y -155.444,Z 1539.276,A 0.000,B 0.000,C 90.000,E1 229.585} C_DIS
LIN {X 0.049,Y -151.763,Z 1539.251,A 0.000,B 0.000,C 90.000,E1 225.081} C_DIS
LIN {X 0.061,Y -149.965,Z 1539.235,A 0.000,B 0.000,C 90.000,E1 222.366} C_DIS
LIN {X -0.028,Y -146.804,Z 1539.210,A 0.000,B 0.000,C 90.000,E1 217.855} C_DIS
LIN {X -0.012,Y -145.380,Z 1539.195,A 0.000,B 0.000,C 90.000,E1 215.105} C_DIS
LIN {X -0.020,Y -142.440,Z 1539.164,A 0.000,B 0.000,C 90.000,E1 209.589} C_DIS
LIN {X 0.027,Y -141.432,Z 1539.149,A 0.000,B 0.000,C 90.000,E1 206.796} C_DIS
LIN {X 0.008,Y -139.366,Z 1539.113,A 0.000,B 0.000,C 90.000,E1 200.301} C_DIS
LIN {X -0.005,Y -138.811,Z 1539.097,A 0.000,B 0.000,C 90.000,E1 197.511} C_DIS
LIN {X 0.045,Y -138.351,Z 1539.056,A 0.000,B 0.000,C 90.000,E1 190.018} C_DIS
LIN {X 0.021,Y -139.540,Z 1539.004,A 0.000,B 0.000,C 90.000,E1 180.688} C_DIS
LIN {X -0.027,Y -141.235,Z 1538.973,A 0.000,B 0.000,C 90.000,E1 175.122} C_DIS
LIN {X -0.068,Y -142.605,Z 1538.957,A 0.000,B 0.000,C 90.000,E1 172.356} C_DIS
LIN {X 0.026,Y -144.915,Z 1538.932,A 0.000,B 0.000,C 90.000,E1 167.701} C_DIS
LIN {X 0.019,Y -147.544,Z 1538.911,A 0.000,B 0.000,C 90.000,E1 164.031} C_DIS
LIN {X 0.051,Y -150.146,Z 1538.891,A 0.000,B 0.000,C 90.000,E1 160.369} C_DIS
LIN {X 0.061,Y -153.514,Z 1538.871,A 0.000,B 0.000,C 90.000,E1 156.741} C_DIS
LIN {X -0.018,Y -157.879,Z 1538.846,A 0.000,B 0.000,C 90.000,E1 152.281} C_DIS
LIN {X -0.063,Y -162.167,Z 1538.826,A 0.000,B 0.000,C 90.000,E1 148.742} C_DIS
LIN {X 0.052,Y -166.374,Z 1538.807,A 0.000,B 0.000,C 90.000,E1 145.182} C_DIS
LIN {X 0.054,Y -171.390,Z 1538.787,A 0.000,B 0.000,C 90.000,E1 141.698} C_DIS
LIN {X 0.094,Y -176.302,Z 1538.768,A 0.000,B 0.000,C 90.000,E1 138.243} C_DIS
LIN {X -0.037,Y -180.589,Z 1538.754,A 0.000,B 0.000,C 90.000,E1 135.729} C_DIS
LIN {X -0.059,Y -185.991,Z 1538.735,A 0.000,B 0.000,C 90.000,E1 132.366} C_DIS
LIN {X -0.004,Y -190.624,Z 1538.721,A 0.000,B 0.000,C 90.000,E1 129.850} C_DIS
LIN {X -0.097,Y -196.375,Z 1538.703,A 0.000,B 0.000,C 90.000,E1 126.583} C_DIS
LIN {X -0.021,Y -201.166,Z 1538.690,A 0.000,B 0.000,C 90.000,E1 124.119} C_DIS
LIN {X 0.046,Y -202.931,Z 1538.684,A 0.000,B 0.000,C 90.000,E1 123.086} C_DIS
LIN {X 0.037,Y -318.253,Z 1538.684,A 0.000,B 0.000,C 90.000,E1 123.086} C_DIS
LIN {X 0.113,Y -320.187,Z 1538.684,A 0.000,B 0.000,C 90.000,E1 123.038} C_DIS
LIN {X 0.150,Y -325.566,Z 1538.682,A 0.000,B 0.000,C 90.000,E1 122.752} C_DIS
LIN {X 0.010,Y -328.448,Z 1538.681,A 0.000,B 0.000,C 90.000,E1 122.498} C_DIS
LIN {X -0.002,Y -332.092,Z 1538.677,A 0.000,B 0.000,C 90.000,E1 121.957} C_DIS
LIN {X -0.172,Y -333.562,Z 1538.676,A 0.000,B 0.000,C 90.000,E1 121.671} C_DIS
LIN {X -0.150,Y -346.138,Z 1538.659,A 0.000,B 0.000,C 90.000,E1 118.565} C_DIS
LIN {X 0.065,Y -358.917,Z 1538.643,A 0.000,B 0.000,C 90.000,E1 115.796} C_DIS
LIN {X 0.008,Y -373.211,Z 1538.629,A 0.000,B 0.000,C 90.000,E1 113.131} C_DIS
LIN {X 0.110,Y -387.291,Z 1538.616,A 0.000,B 0.000,C 90.000,E1 110.791} C_DIS
LIN {X -0.070,Y -402.767,Z 1538.603,A 0.000,B 0.000,C 90.000,E1 108.544} C_DIS
LIN {X -0.002,Y -419.743,Z 1538.591,A 0.000,B 0.000,C 90.000,E1 106.315} C_DIS
LIN {X -0.170,Y -438.340,Z 1538.579,A 0.000,B 0.000,C 90.000,E1 104.175} C_DIS
LIN {X -0.168,Y -458.199,Z 1538.567,A 0.000,B 0.000,C 90.000,E1 102.119} C_DIS
LIN {X 0.090,Y -478.633,Z 1538.557,A 0.000,B 0.000,C 90.000,E1 100.197} C_DIS
LIN {X 0.074,Y -491.660,Z 1538.551,A 0.000,B 0.000,C 90.000,E1 99.095} C_DIS
LIN {X 0.238,Y -493.802,Z 1538.549,A 0.000,B 0.000,C 90.000,E1 98.859} C_DIS
LIN {X -0.088,Y -495.432,Z 1538.548,A 0.000,B 0.000,C 90.000,E1 98.681} C_DIS
LIN {X -0.248,Y -496.839,Z 1538.547,A 0.000,B 0.000,C 90.000,E1 98.454} C_DIS
LIN {X 0.156,Y -497.878,Z 1538.545,A 0.000,B 0.000,C 90.000,E1 98.163} C_DIS
LIN {X -0.073,Y -499.060,Z 1538.543,A 0.000,B 0.000,C 90.000,E1 97.701} C_DIS
LIN {X 0.199,Y -499.210,Z 1538.540,A 0.000,B 0.000,C 90.000,E1 97.182} C_DIS
LIN {X -0.018,Y -498.358,Z 1538.537,A 0.000,B 0.000,C 90.000,E1 96.720} C_DIS
LIN {X -0.231,Y -496.355,Z 1538.535,A 0.000,B 0.000,C 90.000,E1 96.258} C_DIS
LIN {X 0.047,Y -477.393,Z 1538.518,A 0.000,B 0.000,C 90.000,E1 93.269} C_DIS
LIN {X 0.109,Y -469.301,Z 1538.511,A 0.000,B 0.000,C 90.000,E1 92.007} C_DIS
LIN {X -0.159,Y -459.052,Z 1538.503,A 0.000,B 0.000,C 90.000,E1 90.516} C_DIS
LIN {X 0.088,Y -450.141,Z 1538.496,A 0.000,B 0.000,C 90.000,E1 89.198} C_DIS
LIN {X -0.052,Y -439.031,Z 1538.487,A 0.000,B 0.000,C 90.000,E1 87.650} C_DIS
LIN {X 0.050,Y -427.647,Z 1538.478,A 0.000,B 0.000,C 90.000,E1 86.045} C_DIS
LIN {X 0.102,Y -414.291,Z 1538.468,A 0.000,B 0.000,C 90.000,E1 84.147} C_DIS
LIN {X 0.023,Y -399.347,Z 1538.455,A 0.000,B 0.000,C 90.000,E1 81.951} C_DIS
LIN {X 0.128,Y -381.563,Z 1538.440,A 0.000,B 0.000,C 90.000,E1 79.106} C_DIS
LIN {X -0.065,Y -364.780,Z 1538.423,A 0.000,B 0.000,C 90.000,E1 76.228} C_DIS
LIN {X -0.089,Y -351.825,Z 1538.410,A 0.000,B 0.000,C 90.000,E1 73.850} C_DIS
LIN {X 0.103,Y -340.681,Z 1538.398,A 0.000,B 0.000,C 90.000,E1 71.692} C_DIS
LIN {X 0.088,Y -326.718,Z 1538.383,A 0.000,B 0.000,C 90.000,E1 68.901} C_DIS
LIN {X -0.032,Y -312.024,Z 1538.365,A 0.000,B 0.000,C 90.000,E1 65.741} C_DIS
LIN {X -0.002,Y -302.156,Z 1538.353,A 0.000,B 0.000,C 90.000,E1 63.461} C_DIS
LIN {X 0.075,Y -290.898,Z 1538.338,A 0.000,B 0.000,C 90.000,E1 60.795} C_DIS
LIN {X -0.051,Y -281.312,Z 1538.325,A 0.000,B 0.000,C 90.000,E1 58.456} C_DIS
LIN {X 0.085,Y -270.452,Z 1538.309,A 0.000,B 0.000,C 90.000,E1 55.674} C_DIS
LIN {X -0.135,Y -258.740,Z 1538.292,A 0.000,B 0.000,C 90.000,E1 52.557} C_DIS
LIN {X -0.042,Y -247.627,Z 1538.274,A 0.000,B 0.000,C 90.000,E1 49.299} C_DIS
LIN {X 0.040,Y -237.313,Z 1538.255,A 0.000,B 0.000,C 90.000,E1 45.972} C_DIS
LIN {X 0.050,Y -228.898,Z 1538.239,A 0.000,B 0.000,C 90.000,E1 42.975} C_DIS
LIN {X 0.056,Y -221.300,Z 1538.222,A 0.000,B 0.000,C 90.000,E1 39.930} C_DIS
LIN {X -0.061,Y -214.404,Z 1538.205,A 0.000,B 0.000,C 90.000,E1 36.870} C_DIS
LIN {X 0.043,Y -208.302,Z 1538.187,A 0.000,B 0.000,C 90.000,E1 33.706} C_DIS
LIN {X 0.000,Y -202.939,Z 1538.170,A 0.000,B 0.000,C 90.000,E1 30.541} C_DIS
LIN {X 0.106,Y -197.207,Z 1538.147,A 0.000,B 0.000,C 90.000,E1 26.488} C_DIS
LIN {X -0.046,Y -192.321,Z 1538.125,A 0.000,B 0.000,C 90.000,E1 22.461} C_DIS
LIN {X -0.098,Y -188.193,Z 1538.102,A 0.000,B 0.000,C 90.000,E1 18.362} C_DIS
LIN {X -0.029,Y -184.216,Z 1538.074,A 0.000,B 0.000,C 90.000,E1 13.355} C_DIS
LIN {X -0.075,Y -181.191,Z 1538.046,A 0.000,B 0.000,C 90.000,E1 8.341} C_DIS
LIN {X -0.084,Y -178.715,Z 1538.004,A 0.000,B 0.000,C 90.000,E1 0.745} C_DIS
LIN {X 0.033,Y -179.323,Z 1537.955,A 0.000,B 0.000,C 90.000,E1 351.894} C_DIS
LIN {X -0.002,Y -181.765,Z 1537.922,A 0.000,B 0.000,C 90.000,E1 345.992} C_DIS
LIN {X -0.048,Y -185.201,Z 1537.894,A 0.000,B 0.000,C 90.000,E1 340.967} C_DIS
LIN {X -0.027,Y -189.039,Z 1537.871,A 0.000,B 0.000,C 90.000,E1 336.794} C_DIS
LIN {X -0.030,Y -193.901,Z 1537.848,A 0.000,B 0.000,C 90.000,E1 332.666} C_DIS
LIN {X -0.033,Y -199.688,Z 1537.825,A 0.000,B 0.000,C 90.000,E1 328.584} C_DIS
LIN {X 0.021,Y -204.978,Z 1537.807,A 0.000,B 0.000,C 90.000,E1 325.341} C_DIS
LIN {X 0.044,Y -211.053,Z 1537.790,A 0.000,B 0.000,C 90.000,E1 322.145} C_DIS
LIN {X -0.016,Y -217.969,Z 1537.772,A 0.000,B 0.000,C 90.000,E1 319.013} C_DIS
LIN {X -0.003,Y -226.632,Z 1537.753,A 0.000,B 0.000,C 90.000,E1 315.526} C_DIS
LIN {X -0.049,Y -236.429,Z 1537.734,A 0.000,B 0.000,C 90.000,E1 312.123} C_DIS
LIN {X -0.032,Y -242.639,Z 1537.724,A 0.000,B 0.000,C 90.000,E1 310.253} C_DIS
LIN {X 0.087,Y -249.712,Z 1537.713,A 0.000,B 0.000,C 90.000,E1 308.382} C_DIS
LIN {X -0.015,Y -256.067,Z 1537.705,A 0.000,B 0.000,C 90.000,E1 306.950} C_DIS
LIN {X -0.038,Y -263.110,Z 1537.697,A 0.000,B 0.000,C 90.000,E1 305.518} C_DIS
LIN {X 0.087,Y -275.039,Z 1537.686,A 0.000,B 0.000,C 90.000,E1 303.372} C_DIS
LIN {X -0.085,Y -288.539,Z 1537.674,A 0.000,B 0.000,C 90.000,E1 301.337} C_DIS
LIN {X 0.026,Y -310.740,Z 1537.657,A 0.000,B 0.000,C 90.000,E1 298.309} C_DIS
LIN {X 0.083,Y -326.439,Z 1537.646,A 0.000,B 0.000,C 90.000,E1 296.360} C_DIS
LIN {X 0.137,Y -344.778,Z 1537.635,A 0.000,B 0.000,C 90.000,E1 294.207} C_DIS
LIN {X -0.077,Y -363.346,Z 1537.623,A 0.000,B 0.000,C 90.000,E1 292.206} C_DIS
LIN {X 0.011,Y -376.375,Z 1537.615,A 0.000,B 0.000,C 90.000,E1 290.791} C_DIS
LIN {X 0.068,Y -384.145,Z 1537.611,A 0.000,B 0.000,C 90.000,E1 289.939} C_DIS
LIN {X 0.134,Y -391.575,Z 1537.606,A 0.000,B 0.000,C 90.000,E1 289.087} C_DIS
LIN {X 0.128,Y -398.598,Z 1537.601,A 0.000,B 0.000,C 90.000,E1 288.236} C_DIS
LIN {X 0.054,Y -404.955,Z 1537.597,A 0.000,B 0.000,C 90.000,E1 287.402} C_DIS
LIN {X 0.047,Y -410.641,Z 1537.592,A 0.000,B 0.000,C 90.000,E1 286.567} C_DIS
LIN {X 0.090,Y -415.571,Z 1537.588,A 0.000,B 0.000,C 90.000,E1 285.733} C_DIS
LIN {X 0.048,Y -418.420,Z 1537.584,A 0.000,B 0.000,C 90.000,E1 285.190} C_DIS
LIN {X 0.163,Y -421.993,Z 1537.580,A 0.000,B 0.000,C 90.000,E1 284.356} C_DIS
LIN {X -0.207,Y -424.894,Z 1537.575,A 0.000,B 0.000,C 90.000,E1 283.592} C_DIS
LIN {X 0.109,Y -426.343,Z 1537.572,A 0.000,B 0.000,C 90.000,E1 283.008} C_DIS
LIN {X 0.023,Y -427.412,Z 1537.569,A 0.000,B 0.000,C 90.000,E1 282.479} C_DIS
LIN {X -0.055,Y -428.002,Z 1537.566,A 0.000,B 0.000,C 90.000,E1 281.951} C_DIS
LIN {X -0.127,Y -428.172,Z 1537.563,A 0.000,B 0.000,C 90.000,E1 281.422} C_DIS
LIN {X -0.197,Y -427.773,Z 1537.560,A 0.000,B 0.000,C 90.000,E1 280.894} C_DIS
LIN {X 0.152,Y -426.853,Z 1537.557,A 0.000,B 0.000,C 90.000,E1 280.310} C_DIS
LIN {X 0.004,Y -425.322,Z 1537.554,A 0.000,B 0.000,C 90.000,E1 279.792} C_DIS
LIN {X -0.077,Y -423.122,Z 1537.551,A 0.000,B 0.000,C 90.000,E1 279.265} C_DIS
LIN {X 0.178,Y -420.124,Z 1537.548,A 0.000,B 0.000,C 90.000,E1 278.690} C_DIS
LIN {X 0.063,Y -416.320,Z 1537.545,A 0.000,B 0.000,C 90.000,E1 278.163} C_DIS
LIN {X -0.128,Y -411.538,Z 1537.542,A 0.000,B 0.000,C 90.000,E1 277.644} C_DIS
LIN {X 0.098,Y -405.877,Z 1537.539,A 0.000,B 0.000,C 90.000,E1 277.068} C_DIS
LIN {X -0.108,Y -399.889,Z 1537.537,A 0.000,B 0.000,C 90.000,E1 276.606} C_DIS
LIN {X 0.017,Y -393.734,Z 1537.534,A 0.000,B 0.000,C 90.000,E1 276.144} C_DIS
LIN {X -0.003,Y -387.210,Z 1537.532,A 0.000,B 0.000,C 90.000,E1 275.739} C_DIS
LIN {X -0.078,Y -380.702,Z 1537.530,A 0.000,B 0.000,C 90.000,E1 275.391} C_DIS
LIN {X -0.163,Y -370.962,Z 1537.527,A 0.000,B 0.000,C 90.000,E1 274.935} C_DIS
LIN {X -0.061,Y -358.217,Z 1537.524,A 0.000,B 0.000,C 90.000,E1 274.359} C_DIS
LIN {X -0.087,Y -345.502,Z 1537.521,A 0.000,B 0.000,C 90.000,E1 273.841} C_DIS
LIN {X 0.093,Y -335.309,Z 1537.519,A 0.000,B 0.000,C 90.000,E1 273.440} C_DIS
LIN {X 0.000,Y -322.169,Z 1537.517,A 0.000,B 0.000,C 90.000,E1 273.037} C_DIS
LIN {X -0.008,Y -311.655,Z 1537.515,A 0.000,B 0.000,C 90.000,E1 272.751} C_DIS
LIN {X -0.066,Y -300.701,Z 1537.514,A 0.000,B 0.000,C 90.000,E1 272.522} C_DIS
LIN {X 0.118,Y -289.012,Z 1537.513,A 0.000,B 0.000,C 90.000,E1 272.293} C_DIS
LIN {X -0.009,Y -276.955,Z 1537.512,A 0.000,B 0.000,C 90.000,E1 272.178} C_DIS
LIN {X -0.102,Y -261.443,Z 1537.512,A 0.000,B 0.000,C 90.000,E1 272.121} C_DIS
LIN {X 0.079,Y -181.247,Z 1537.512,A 0.000,B 0.000,C 90.000,E1 272.064} C_DIS
LIN {X -0.054,Y -181.577,Z 1537.502,A 0.000,B 0.000,C 90.000,E1 270.401} C_DIS
LIN {X -0.077,Y -180.905,Z 1537.474,A 0.000,B 0.000,C 90.000,E1 265.355} C_DIS
LIN {X -0.004,Y -180.669,Z 1537.469,A 0.000,B 0.000,C 90.000,E1 264.489} C_DIS
LIN {X 0.071,Y -178.750,Z 1537.441,A 0.000,B 0.000,C 90.000,E1 259.398} C_DIS
LIN {X -0.032,Y -175.798,Z 1537.413,A 0.000,B 0.000,C 90.000,E1 254.338} C_DIS
LIN {X -0.037,Y -171.983,Z 1537.384,A 0.000,B 0.000,C 90.000,E1 249.209} C_DIS
LIN {X 0.001,Y -171.389,Z 1537.380,A 0.000,B 0.000,C 90.000,E1 248.337} C_DIS
LIN {X -0.014,Y -167.632,Z 1537.356,A 0.000,B 0.000,C 90.000,E1 244.024} C_DIS
LIN {X 0.002,Y -166.289,Z 1537.346,A 0.000,B 0.000,C 90.000,E1 242.281} C_DIS
LIN {X -0.004,Y -163.036,Z 1537.327,A 0.000,B 0.000,C 90.000,E1 238.791} C_DIS
LIN {X -0.042,Y -160.967,Z 1537.312,A 0.000,B 0.000,C 90.000,E1 236.167} C_DIS
LIN {X -0.064,Y -157.719,Z 1537.292,A 0.000,B 0.000,C 90.000,E1 232.637} C_DIS
LIN {X 0.094,Y -155.759,Z 1537.277,A 0.000,B 0.000,C 90.000,E1 229.908} C_DIS
LIN {X -0.070,Y -152.014,Z 1537.253,A 0.000,B 0.000,C 90.000,E1 225.486} C_DIS
LIN {X -0.052,Y -150.261,Z 1537.238,A 0.000,B 0.000,C 90.000,E1 222.771} C_DIS
LIN {X -0.033,Y -147.015,Z 1537.212,A 0.000,B 0.000,C 90.000,E1 218.222} C_DIS
LIN {X -0.012,Y -145.599,Z 1537.197,A 0.000,B 0.000,C 90.000,E1 215.471} C_DIS
LIN {X -0.008,Y -142.985,Z 1537.172,A 0.000,B 0.000,C 90.000,E1 210.875} C_DIS
LIN {X -0.008,Y -141.612,Z 1537.151,A 0.000,B 0.000,C 90.000,E1 207.180} C_DIS
LIN {X 0.034,Y -139.427,Z 1537.115,A 0.000,B 0.000,C 90.000,E1 200.663} C_DIS
LIN {X 0.085,Y -139.157,Z 1537.104,A 0.000,B 0.000,C 90.000,E1 198.779} C_DIS
LIN {X -0.030,Y -138.342,Z 1537.058,A 0.000,B 0.000,C 90.000,E1 190.423} C_DIS
LIN {X -0.048,Y -139.481,Z 1537.006,A 0.000,B 0.000,C 90.000,E1 181.088} C_DIS
LIN {X 0.033,Y -141.073,Z 1536.975,A 0.000,B 0.000,C 90.000,E1 175.469} C_DIS
LIN {X -0.013,Y -142.449,Z 1536.959,A 0.000,B 0.000,C 90.000,E1 172.704} C_DIS
LIN {X 0.077,Y -144.690,Z 1536.934,A 0.000,B 0.000,C 90.000,E1 168.049} C_DIS
LIN {X 0.030,Y -147.282,Z 1536.913,A 0.000,B 0.000,C 90.000,E1 164.393} C_DIS
LIN {X 0.046,Y -150.601,Z 1536.888,A 0.000,B 0.000,C 90.000,E1 159.826} C_DIS
LIN {X -0.018,Y -154.075,Z 1536.868,A 0.000,B 0.000,C 90.000,E1 156.230} C_DIS
LIN {X 0.049,Y -157.494,Z 1536.848,A 0.000,B 0.000,C 90.000,E1 152.615} C_DIS
LIN {X -0.006,Y -161.721,Z 1536.828,A 0.000,B 0.000,C 90.000,E1 149.076} C_DIS
LIN {X 0.007,Y -165.915,Z 1536.809,A 0.000,B 0.000,C 90.000,E1 145.548} C_DIS
LIN {X -0.006,Y -170.902,Z 1536.789,A 0.000,B 0.000,C 90.000,E1 142.065} C_DIS
LIN {X 0.021,Y -175.770,Z 1536.770,A 0.000,B 0.000,C 90.000,E1 138.609} C_DIS
LIN {X 0.022,Y -181.380,Z 1536.751,A 0.000,B 0.000,C 90.000,E1 135.202} C_DIS
LIN {X 0.026,Y -186.874,Z 1536.732,A 0.000,B 0.000,C 90.000,E1 131.838} C_DIS
LIN {X -0.021,Y -191.459,Z 1536.719,A 0.000,B 0.000,C 90.000,E1 129.358} C_DIS
LIN {X -0.090,Y -197.314,Z 1536.700,A 0.000,B 0.000,C 90.000,E1 126.091} C_DIS
LIN {X -0.053,Y -200.591,Z 1536.691,A 0.000,B 0.000,C 90.000,E1 124.452} C_DIS
LIN {X -0.110,Y -202.868,Z 1536.684,A 0.000,B 0.000,C 90.000,E1 123.166} C_DIS
LIN {X 0.046,Y -318.333,Z 1536.684,A 0.000,B 0.000,C 90.000,E1 123.118} C_DIS
LIN {X 0.078,Y -319.777,Z 1536.684,A 0.000,B 0.000,C 90.000,E1 123.086} C_DIS
LIN {X -0.058,Y -325.316,Z 1536.682,A 0.000,B 0.000,C 90.000,E1 122.832} C_DIS
LIN {X 0.080,Y -328.488,Z 1536.681,A 0.000,B 0.000,C 90.000,E1 122.498} C_DIS
LIN {X 0.050,Y -332.074,Z 1536.678,A 0.000,B 0.000,C 90.000,E1 121.957} C_DIS
LIN {X -0.120,Y -333.515,Z 1536.676,A 0.000,B 0.000,C 90.000,E1 121.671} C_DIS
LIN {X -0.096,Y -346.078,Z 1536.659,A 0.000,B 0.000,C 90.000,E1 118.565} C_DIS
LIN {X 0.118,Y -358.853,Z 1536.643,A 0.000,B 0.000,C 90.000,E1 115.796} C_DIS
LIN {X 0.061,Y -373.140,Z 1536.629,A 0.000,B 0.000,C 90.000,E1 113.131} C_DIS
LIN {X 0.163,Y -387.216,Z 1536.616,A 0.000,B 0.000,C 90.000,E1 110.791} C_DIS
LIN {X -0.017,Y -402.685,Z 1536.603,A 0.000,B 0.000,C 90.000,E1 108.544} C_DIS
LIN {X 0.052,Y -419.657,Z 1536.591,A 0.000,B 0.000,C 90.000,E1 106.315} C_DIS
LIN {X -0.116,Y -438.248,Z 1536.579,A 0.000,B 0.000,C 90.000,E1 104.175} C_DIS
LIN {X -0.116,Y -458.105,Z 1536.567,A 0.000,B 0.000,C 90.000,E1 102.119} C_DIS
LIN {X 0.138,Y -478.537,Z 1536.557,A 0.000,B 0.000,C 90.000,E1 100.197} C_DIS
LIN {X 0.120,Y -491.562,Z 1536.551,A 0.000,B 0.000,C 90.000,E1 99.095} C_DIS
LIN {X -0.204,Y -493.703,Z 1536.549,A 0.000,B 0.000,C 90.000,E1 98.916} C_DIS
LIN {X -0.042,Y -495.332,Z 1536.548,A 0.000,B 0.000,C 90.000,E1 98.681} C_DIS
LIN {X -0.203,Y -496.737,Z 1536.547,A 0.000,B 0.000,C 90.000,E1 98.454} C_DIS
LIN {X 0.201,Y -497.775,Z 1536.546,A 0.000,B 0.000,C 90.000,E1 98.163} C_DIS
LIN {X -0.028,Y -498.956,Z 1536.543,A 0.000,B 0.000,C 90.000,E1 97.701} C_DIS
LIN {X -0.252,Y -499.106,Z 1536.540,A 0.000,B 0.000,C 90.000,E1 97.239} C_DIS
LIN {X 0.026,Y -498.252,Z 1536.537,A 0.000,B 0.000,C 90.000,E1 96.720} C_DIS
LIN {X -0.190,Y -496.249,Z 1536.535,A 0.000,B 0.000,C 90.000,E1 96.258} C_DIS
LIN {X 0.085,Y -477.312,Z 1536.518,A 0.000,B 0.000,C 90.000,E1 93.269} C_DIS
LIN {X -0.135,Y -470.886,Z 1536.513,A 0.000,B 0.000,C 90.000,E1 92.293} C_DIS
LIN {X 0.088,Y -460.718,Z 1536.504,A 0.000,B 0.000,C 90.000,E1 90.745} C_DIS
LIN {X -0.101,Y -451.866,Z 1536.497,A 0.000,B 0.000,C 90.000,E1 89.484} C_DIS
LIN {X -0.206,Y -440.840,Z 1536.488,A 0.000,B 0.000,C 90.000,E1 87.936} C_DIS
LIN {X -0.063,Y -429.524,Z 1536.480,A 0.000,B 0.000,C 90.000,E1 86.331} C_DIS
LIN {X 0.129,Y -414.332,Z 1536.468,A 0.000,B 0.000,C 90.000,E1 84.147} C_DIS
LIN {X 0.051,Y -399.399,Z 1536.455,A 0.000,B 0.000,C 90.000,E1 81.951} C_DIS
LIN {X 0.155,Y -381.597,Z 1536.440,A 0.000,B 0.000,C 90.000,E1 79.106} C_DIS
LIN {X -0.021,Y -366.466,Z 1536.425,A 0.000,B 0.000,C 90.000,E1 76.520} C_DIS
LIN {X -0.100,Y -353.466,Z 1536.412,A 0.000,B 0.000,C 90.000,E1 74.157} C_DIS
LIN {X 0.118,Y -342.313,Z 1536.400,A 0.000,B 0.000,C 90.000,E1 72.000} C_DIS
LIN {X 0.148,Y -328.267,Z 1536.385,A 0.000,B 0.000,C 90.000,E1 69.209} C_DIS
LIN {X 0.140,Y -314.938,Z 1536.369,A 0.000,B 0.000,C 90.000,E1 66.357} C_DIS
LIN {X 0.129,Y -303.610,Z 1536.354,A 0.000,B 0.000,C 90.000,E1 63.768} C_DIS
LIN {X -0.154,Y -293.747,Z 1536.342,A 0.000,B 0.000,C 90.000,E1 61.513} C_DIS
LIN {X 0.009,Y -282.754,Z 1536.327,A 0.000,B 0.000,C 90.000,E1 58.791} C_DIS
LIN {X 0.089,Y -273.249,Z 1536.313,A 0.000,B 0.000,C 90.000,E1 56.373} C_DIS
LIN {X -0.002,Y -260.125,Z 1536.294,A 0.000,B 0.000,C 90.000,E1 52.889} C_DIS
LIN {X -0.023,Y -248.963,Z 1536.276,A 0.000,B 0.000,C 90.000,E1 49.666} C_DIS
LIN {X -0.068,Y -238.572,Z 1536.258,A 0.000,B 0.000,C 90.000,E1 46.377} C_DIS
LIN {X -0.060,Y -229.115,Z 1536.239,A 0.000,B 0.000,C 90.000,E1 43.014} C_DIS
LIN {X 0.105,Y -221.531,Z 1536.222,A 0.000,B 0.000,C 90.000,E1 39.930} C_DIS
LIN {X -0.007,Y -214.680,Z 1536.205,A 0.000,B 0.000,C 90.000,E1 36.870} C_DIS
LIN {X 0.102,Y -208.611,Z 1536.187,A 0.000,B 0.000,C 90.000,E1 33.706} C_DIS
LIN {X 0.064,Y -203.255,Z 1536.170,A 0.000,B 0.000,C 90.000,E1 30.541} C_DIS
LIN {X 0.002,Y -197.518,Z 1536.147,A 0.000,B 0.000,C 90.000,E1 26.539} C_DIS
LIN {X 0.035,Y -192.597,Z 1536.125,A 0.000,B 0.000,C 90.000,E1 22.461} C_DIS
LIN {X -0.012,Y -188.471,Z 1536.102,A 0.000,B 0.000,C 90.000,E1 18.362} C_DIS
LIN {X 0.066,Y -184.505,Z 1536.074,A 0.000,B 0.000,C 90.000,E1 13.355} C_DIS
LIN {X 0.029,Y -181.476,Z 1536.046,A 0.000,B 0.000,C 90.000,E1 8.341} C_DIS
LIN {X 0.034,Y -178.973,Z 1536.004,A 0.000,B 0.000,C 90.000,E1 0.745} C_DIS
LIN {X 0.048,Y -179.600,Z 1535.955,A 0.000,B 0.000,C 90.000,E1 351.894} C_DIS
LIN {X 0.024,Y -182.012,Z 1535.922,A 0.000,B 0.000,C 90.000,E1 345.992} C_DIS
LIN {X -0.011,Y -185.452,Z 1535.894,A 0.000,B 0.000,C 90.000,E1 340.967} C_DIS
LIN {X 0.017,Y -189.256,Z 1535.871,A 0.000,B 0.000,C 90.000,E1 336.794} C_DIS
LIN {X 0.023,Y -194.100,Z 1535.848,A 0.000,B 0.000,C 90.000,E1 332.666} C_DIS
LIN {X 0.028,Y -199.860,Z 1535.826,A 0.000,B 0.000,C 90.000,E1 328.584} C_DIS
LIN {X -0.081,Y -205.136,Z 1535.808,A 0.000,B 0.000,C 90.000,E1 325.388} C_DIS
LIN {X -0.050,Y -211.176,Z 1535.790,A 0.000,B 0.000,C 90.000,E1 322.190} C_DIS
LIN {X 0.063,Y -218.064,Z 1535.772,A 0.000,B 0.000,C 90.000,E1 319.013} C_DIS
LIN {X -0.082,Y -226.715,Z 1535.753,A 0.000,B 0.000,C 90.000,E1 315.567} C_DIS
LIN {X 0.041,Y -236.487,Z 1535.734,A 0.000,B 0.000,C 90.000,E1 312.123} C_DIS
LIN {X 0.060,Y -242.682,Z 1535.724,A 0.000,B 0.000,C 90.000,E1 310.253} C_DIS
LIN {X 0.028,Y -249.714,Z 1535.714,A 0.000,B 0.000,C 90.000,E1 308.418} C_DIS
LIN {X 0.112,Y -257.673,Z 1535.703,A 0.000,B 0.000,C 90.000,E1 306.583} C_DIS
LIN {X -0.042,Y -264.893,Z 1535.695,A 0.000,B 0.000,C 90.000,E1 305.185} C_DIS
LIN {X -0.038,Y -274.910,Z 1535.686,A 0.000,B 0.000,C 90.000,E1 303.420} C_DIS
LIN {X 0.021,Y -288.346,Z 1535.674,A 0.000,B 0.000,C 90.000,E1 301.337} C_DIS
LIN {X -0.139,Y -310.541,Z 1535.657,A 0.000,B 0.000,C 90.000,E1 298.359} C_DIS
LIN {X -0.098,Y -326.304,Z 1535.647,A 0.000,B 0.000,C 90.000,E1 296.411} C_DIS
LIN {X 0.153,Y -344.854,Z 1535.635,A 0.000,B 0.000,C 90.000,E1 294.207} C_DIS
LIN {X 0.031,Y -361.017,Z 1535.625,A 0.000,B 0.000,C 90.000,E1 292.461} C_DIS
LIN {X 0.056,Y -374.196,Z 1535.617,A 0.000,B 0.000,C 90.000,E1 291.046} C_DIS
LIN {X -0.075,Y -384.582,Z 1535.611,A 0.000,B 0.000,C 90.000,E1 289.939} C_DIS
LIN {X -0.067,Y -392.071,Z 1535.606,A 0.000,B 0.000,C 90.000,E1 289.087} C_DIS
LIN {X -0.073,Y -399.087,Z 1535.601,A 0.000,B 0.000,C 90.000,E1 288.236} C_DIS
LIN {X -0.146,Y -405.454,Z 1535.597,A 0.000,B 0.000,C 90.000,E1 287.402} C_DIS
LIN {X -0.032,Y -411.113,Z 1535.592,A 0.000,B 0.000,C 90.000,E1 286.551} C_DIS
LIN {X 0.007,Y -416.041,Z 1535.587,A 0.000,B 0.000,C 90.000,E1 285.717} C_DIS
LIN {X -0.010,Y -420.161,Z 1535.583,A 0.000,B 0.000,C 90.000,E1 284.898} C_DIS
LIN {X -0.028,Y -422.531,Z 1535.580,A 0.000,B 0.000,C 90.000,E1 284.356} C_DIS
LIN {X 0.018,Y -425.376,Z 1535.575,A 0.000,B 0.000,C 90.000,E1 283.536} C_DIS
LIN {X -0.077,Y -426.843,Z 1535.572,A 0.000,B 0.000,C 90.000,E1 283.008} C_DIS
LIN {X -0.161,Y -427.888,Z 1535.569,A 0.000,B 0.000,C 90.000,E1 282.479} C_DIS
LIN {X -0.236,Y -428.499,Z 1535.566,A 0.000,B 0.000,C 90.000,E1 281.951} C_DIS
LIN {X 0.115,Y -428.620,Z 1535.563,A 0.000,B 0.000,C 90.000,E1 281.366} C_DIS
LIN {X 0.048,Y -428.264,Z 1535.560,A 0.000,B 0.000,C 90.000,E1 280.838} C_DIS
LIN {X -0.020,Y -427.350,Z 1535.557,A 0.000,B 0.000,C 90.000,E1 280.310} C_DIS
LIN {X -0.164,Y -425.819,Z 1535.554,A 0.000,B 0.000,C 90.000,E1 279.792} C_DIS
LIN {X 0.177,Y -423.647,Z 1535.551,A 0.000,B 0.000,C 90.000,E1 279.208} C_DIS
LIN {X 0.087,Y -420.673,Z 1535.548,A 0.000,B 0.000,C 90.000,E1 278.681} C_DIS
LIN {X -0.087,Y -416.825,Z 1535.545,A 0.000,B 0.000,C 90.000,E1 278.163} C_DIS
LIN {X 0.135,Y -412.016,Z 1535.542,A 0.000,B 0.000,C 90.000,E1 277.587} C_DIS
LIN {X -0.040,Y -406.342,Z 1535.539,A 0.000,B 0.000,C 90.000,E1 277.068} C_DIS
LIN {X 0.170,Y -400.287,Z 1535.536,A 0.000,B 0.000,C 90.000,E1 276.549} C_DIS
LIN {X -0.036,Y -394.261,Z 1535.534,A 0.000,B 0.000,C 90.000,E1 276.144} C_DIS
LIN {X 0.017,Y -387.919,Z 1535.532,A 0.000,B 0.000,C 90.000,E1 275.739} C_DIS
LIN {X -0.045,Y -381.453,Z 1535.530,A 0.000,B 0.000,C 90.000,E1 275.391} C_DIS
LIN {X -0.131,Y -371.741,Z 1535.527,A 0.000,B 0.000,C 90.000,E1 274.935} C_DIS
LIN {X -0.132,Y -355.807,Z 1535.523,A 0.000,B 0.000,C 90.000,E1 274.245} C_DIS
LIN {X -0.082,Y -343.145,Z 1535.521,A 0.000,B 0.000,C 90.000,E1 273.726} C_DIS
LIN {X -0.148,Y -332.813,Z 1535.519,A 0.000,B 0.000,C 90.000,E1 273.383} C_DIS
LIN {X 0.153,Y -319.763,Z 1535.516,A 0.000,B 0.000,C 90.000,E1 272.922} C_DIS
LIN {X 0.090,Y -313.036,Z 1535.515,A 0.000,B 0.000,C 90.000,E1 272.751} C_DIS
LIN {X 0.041,Y -302.213,Z 1535.514,A 0.000,B 0.000,C 90.000,E1 272.522} C_DIS
LIN {X -0.101,Y -290.426,Z 1535.513,A 0.000,B 0.000,C 90.000,E1 272.350} C_DIS
LIN {X -0.093,Y -282.056,Z 1535.512,A 0.000,B 0.000,C 90.000,E1 272.236} C_DIS
LIN {X -0.005,Y -267.358,Z 1535.512,A 0.000,B 0.000,C 90.000,E1 272.121} C_DIS
LIN {X -0.103,Y -257.524,Z 1535.512,A 0.000,B 0.000,C 90.000,E1 272.121} C_DIS
LIN {X 0.073,Y -181.247,Z 1535.512,A 0.000,B 0.000,C 90.000,E1 272.064} C_DIS
LIN {X -0.005,Y -181.568,Z 1535.500,A 0.000,B 0.000,C 90.000,E1 270.057} C_DIS
LIN {X -0.017,Y -180.863,Z 1535.472,A 0.000,B 0.000,C 90.000,E1 265.008} C_DIS
LIN {X 0.037,Y -178.976,Z 1535.444,A 0.000,B 0.000,C 90.000,E1 259.926} C_DIS
LIN {X 0.047,Y -177.940,Z 1535.435,A 0.000,B 0.000,C 90.000,E1 258.229} C_DIS
LIN {X 0.062,Y -175.579,Z 1535.411,A 0.000,B 0.000,C 90.000,E1 253.976} C_DIS
LIN {X 0.068,Y -172.306,Z 1535.387,A 0.000,B 0.000,C 90.000,E1 249.699} C_DIS
LIN {X 0.045,Y -171.785,Z 1535.383,A 0.000,B 0.000,C 90.000,E1 248.847} C_DIS
LIN {X -0.077,Y -169.451,Z 1535.368,A 0.000,B 0.000,C 90.000,E1 246.305} C_DIS
LIN {X -0.021,Y -166.781,Z 1535.349,A 0.000,B 0.000,C 90.000,E1 242.820} C_DIS
LIN {X -0.024,Y -162.761,Z 1535.325,A 0.000,B 0.000,C 90.000,E1 238.456} C_DIS
LIN {X -0.049,Y -161.451,Z 1535.315,A 0.000,B 0.000,C 90.000,E1 236.707} C_DIS
LIN {X -0.007,Y -157.444,Z 1535.290,A 0.000,B 0.000,C 90.000,E1 232.271} C_DIS
LIN {X 0.027,Y -155.453,Z 1535.276,A 0.000,B 0.000,C 90.000,E1 229.585} C_DIS
LIN {X 0.075,Y -151.769,Z 1535.251,A 0.000,B 0.000,C 90.000,E1 225.081} C_DIS
LIN {X -0.015,Y -149.973,Z 1535.236,A 0.000,B 0.000,C 90.000,E1 222.405} C_DIS
LIN {X -0.003,Y -146.809,Z 1535.210,A 0.000,B 0.000,C 90.000,E1 217.855} C_DIS
LIN {X 0.013,Y -145.388,Z 1535.195,A 0.000,B 0.000,C 90.000,E1 215.105} C_DIS
LIN {X 0.004,Y -142.825,Z 1535.170,A 0.000,B 0.000,C 90.000,E1 210.512} C_DIS
LIN {X -0.013,Y -141.438,Z 1535.149,A 0.000,B 0.000,C 90.000,E1 206.821} C_DIS
LIN {X 0.033,Y -139.368,Z 1535.113,A 0.000,B 0.000,C 90.000,E1 200.301} C_DIS
LIN {X 0.018,Y -138.813,Z 1535.097,A 0.000,B 0.000,C 90.000,E1 197.511} C_DIS
LIN {X 0.069,Y -138.351,Z 1535.056,A 0.000,B 0.000,C 90.000,E1 190.018} C_DIS
LIN {X 0.045,Y -139.539,Z 1535.004,A 0.000,B 0.000,C 90.000,E1 180.688} C_DIS
LIN {X -0.002,Y -141.231,Z 1534.973,A 0.000,B 0.000,C 90.000,E1 175.122} C_DIS
LIN {X -0.043,Y -142.602,Z 1534.957,A 0.000,B 0.000,C 90.000,E1 172.356} C_DIS
LIN {X 0.052,Y -144.910,Z 1534.932,A 0.000,B 0.000,C 90.000,E1 167.701} C_DIS
LIN {X 0.044,Y -147.538,Z 1534.911,A 0.000,B 0.000,C 90.000,E1 164.031} C_DIS
LIN {X -0.064,Y -150.137,Z 1534.891,A 0.000,B 0.000,C 90.000,E1 160.423} C_DIS
LIN {X -0.054,Y -153.504,Z 1534.871,A 0.000,B 0.000,C 90.000,E1 156.794} C_DIS
LIN {X 0.008,Y -157.869,Z 1534.846,A 0.000,B 0.000,C 90.000,E1 152.281} C_DIS
LIN {X -0.036,Y -162.155,Z 1534.826,A 0.000,B 0.000,C 90.000,E1 148.742} C_DIS
LIN {X 0.079,Y -166.362,Z 1534.807,A 0.000,B 0.000,C 90.000,E1 145.182} C_DIS
LIN {X -0.052,Y -171.378,Z 1534.787,A 0.000,B 0.000,C 90.000,E1 141.743} C_DIS
LIN {X -0.009,Y -176.288,Z 1534.768,A 0.000,B 0.000,C 90.000,E1 138.286} C_DIS
LIN {X -0.008,Y -180.574,Z 1534.754,A 0.000,B 0.000,C 90.000,E1 135.729} C_DIS
LIN {X -0.030,Y -185.975,Z 1534.735,A 0.000,B 0.000,C 90.000,E1 132.366} C_DIS
LIN {X 0.025,Y -190.608,Z 1534.721,A 0.000,B 0.000,C 90.000,E1 129.850} C_DIS
LIN {X -0.067,Y -196.358,Z 1534.703,A 0.000,B 0.000,C 90.000,E1 126.583} C_DIS
LIN {X 0.010,Y -201.152,Z 1534.690,A 0.000,B 0.000,C 90.000,E1 124.119} C_DIS
LIN {X 0.013,Y -202.806,Z 1534.684,A 0.000,B 0.000,C 90.000,E1 123.166} C_DIS
LIN {X -0.016,Y -318.092,Z 1534.684,A 0.000,B 0.000,C 90.000,E1 123.166} C_DIS
LIN {X -0.214,Y -319.972,Z 1534.684,A 0.000,B 0.000,C 90.000,E1 123.166} C_DIS
LIN {X -0.079,Y -325.657,Z 1534.682,A 0.000,B 0.000,C 90.000,E1 122.832} C_DIS
LIN {X 0.061,Y -328.658,Z 1534.681,A 0.000,B 0.000,C 90.000,E1 122.498} C_DIS
LIN {X 0.068,Y -330.661,Z 1534.679,A 0.000,B 0.000,C 90.000,E1 122.212} C_DIS
LIN {X 0.074,Y -332.230,Z 1534.677,A 0.000,B 0.000,C 90.000,E1 121.926} C_DIS
LIN {X -0.146,Y -334.785,Z 1534.674,A 0.000,B 0.000,C 90.000,E1 121.337} C_DIS
LIN {X -0.074,Y -346.159,Z 1534.658,A 0.000,B 0.000,C 90.000,E1 118.537} C_DIS
LIN {X -0.026,Y -358.945,Z 1534.643,A 0.000,B 0.000,C 90.000,E1 115.796} C_DIS
LIN {X -0.087,Y -373.246,Z 1534.628,A 0.000,B 0.000,C 90.000,E1 113.131} C_DIS
LIN {X 0.012,Y -387.335,Z 1534.615,A 0.000,B 0.000,C 90.000,E1 110.791} C_DIS
LIN {X -0.170,Y -402.819,Z 1534.603,A 0.000,B 0.000,C 90.000,E1 108.544} C_DIS
LIN {X -0.105,Y -419.805,Z 1534.591,A 0.000,B 0.000,C 90.000,E1 106.315} C_DIS
LIN {X 0.149,Y -438.411,Z 1534.578,A 0.000,B 0.000,C 90.000,E1 104.120} C_DIS
LIN {X 0.175,Y -458.275,Z 1534.567,A 0.000,B 0.000,C 90.000,E1 102.063} C_DIS
LIN {X -0.013,Y -478.713,Z 1534.557,A 0.000,B 0.000,C 90.000,E1 100.197} C_DIS
LIN {X -0.027,Y -491.720,Z 1534.551,A 0.000,B 0.000,C 90.000,E1 99.095} C_DIS
LIN {X 0.128,Y -493.803,Z 1534.549,A 0.000,B 0.000,C 90.000,E1 98.859} C_DIS
LIN {X -0.208,Y -495.391,Z 1534.548,A 0.000,B 0.000,C 90.000,E1 98.681} C_DIS
LIN {X 0.122,Y -496.754,Z 1534.547,A 0.000,B 0.000,C 90.000,E1 98.398} C_DIS
LIN {X 0.035,Y -497.758,Z 1534.545,A 0.000,B 0.000,C 90.000,E1 98.163} C_DIS
LIN {X -0.195,Y -498.882,Z 1534.543,A 0.000,B 0.000,C 90.000,E1 97.701} C_DIS
LIN {X 0.076,Y -498.981,Z 1534.540,A 0.000,B 0.000,C 90.000,E1 97.182} C_DIS
LIN {X -0.141,Y -498.074,Z 1534.537,A 0.000,B 0.000,C 90.000,E1 96.720} C_DIS
LIN {X 0.137,Y -496.004,Z 1534.535,A 0.000,B 0.000,C 90.000,E1 96.201} C_DIS
LIN {X -0.222,Y -480.165,Z 1534.521,A 0.000,B 0.000,C 90.000,E1 93.784} C_DIS
LIN {X -0.121,Y -472.302,Z 1534.514,A 0.000,B 0.000,C 90.000,E1 92.522} C_DIS
LIN {X 0.125,Y -462.205,Z 1534.505,A 0.000,B 0.000,C 90.000,E1 90.974} C_DIS
LIN {X -0.040,Y -453.424,Z 1534.498,A 0.000,B 0.000,C 90.000,E1 89.714} C_DIS
LIN {X -0.120,Y -442.450,Z 1534.490,A 0.000,B 0.000,C 90.000,E1 88.165} C_DIS
LIN {X 0.052,Y -431.181,Z 1534.481,A 0.000,B 0.000,C 90.000,E1 86.560} C_DIS
LIN {X 0.145,Y -417.922,Z 1534.470,A 0.000,B 0.000,C 90.000,E1 84.666} C_DIS
LIN {X 0.148,Y -402.943,Z 1534.458,A 0.000,B 0.000,C 90.000,E1 82.470} C_DIS
LIN {X -0.087,Y -384.903,Z 1534.443,A 0.000,B 0.000,C 90.000,E1 79.690} C_DIS
LIN {X 0.106,Y -371.327,Z 1534.430,A 0.000,B 0.000,C 90.000,E1 77.353} C_DIS
LIN {X 0.131,Y -358.195,Z 1534.417,A 0.000,B 0.000,C 90.000,E1 74.991} C_DIS
LIN {X 0.035,Y -345.373,Z 1534.403,A 0.000,B 0.000,C 90.000,E1 72.598} C_DIS
LIN {X 0.058,Y -332.760,Z 1534.390,A 0.000,B 0.000,C 90.000,E1 70.134} C_DIS
LIN {X 0.059,Y -316.307,Z 1534.370,A 0.000,B 0.000,C 90.000,E1 66.666} C_DIS
LIN {X -0.015,Y -303.513,Z 1534.354,A 0.000,B 0.000,C 90.000,E1 63.768} C_DIS
LIN {X 0.103,Y -293.672,Z 1534.341,A 0.000,B 0.000,C 90.000,E1 61.435} C_DIS
LIN {X 0.111,Y -282.698,Z 1534.326,A 0.000,B 0.000,C 90.000,E1 58.742} C_DIS
LIN {X -0.046,Y -273.217,Z 1534.313,A 0.000,B 0.000,C 90.000,E1 56.373} C_DIS
LIN {X 0.077,Y -260.119,Z 1534.294,A 0.000,B 0.000,C 90.000,E1 52.844} C_DIS
LIN {X 0.044,Y -248.987,Z 1534.276,A 0.000,B 0.000,C 90.000,E1 49.622} C_DIS
LIN {X -0.021,Y -238.634,Z 1534.257,A 0.000,B 0.000,C 90.000,E1 46.338} C_DIS
LIN {X -0.014,Y -229.232,Z 1534.239,A 0.000,B 0.000,C 90.000,E1 42.975} C_DIS
LIN {X 0.001,Y -221.672,Z 1534.222,A 0.000,B 0.000,C 90.000,E1 39.930} C_DIS
LIN {X -0.105,Y -214.871,Z 1534.205,A 0.000,B 0.000,C 90.000,E1 36.870} C_DIS
LIN {X 0.013,Y -208.832,Z 1534.187,A 0.000,B 0.000,C 90.000,E1 33.706} C_DIS
LIN {X -0.026,Y -202.282,Z 1534.165,A 0.000,B 0.000,C 90.000,E1 29.745} C_DIS
LIN {X -0.033,Y -196.731,Z 1534.143,A 0.000,B 0.000,C 90.000,E1 25.720} C_DIS
LIN {X -0.026,Y -191.946,Z 1534.120,A 0.000,B 0.000,C 90.000,E1 21.642} C_DIS
LIN {X 0.016,Y -187.984,Z 1534.097,A 0.000,B 0.000,C 90.000,E1 17.511} C_DIS
LIN {X -0.022,Y -184.165,Z 1534.070,A 0.000,B 0.000,C 90.000,E1 12.535} C_DIS
LIN {X -0.017,Y -180.952,Z 1534.037,A 0.000,B 0.000,C 90.000,E1 6.663} C_DIS
LIN {X 0.053,Y -179.047,Z 1533.988,A 0.000,B 0.000,C 90.000,E1 357.822} C_DIS
LIN {X -0.047,Y -180.102,Z 1533.950,A 0.000,B 0.000,C 90.000,E1 351.084} C_DIS
LIN {X -0.017,Y -182.757,Z 1533.918,A 0.000,B 0.000,C 90.000,E1 345.172} C_DIS
LIN {X 0.018,Y -186.377,Z 1533.890,A 0.000,B 0.000,C 90.000,E1 340.134} C_DIS
LIN {X 0.037,Y -190.374,Z 1533.867,A 0.000,B 0.000,C 90.000,E1 335.973} C_DIS
LIN {X -0.098,Y -195.374,Z 1533.844,A 0.000,B 0.000,C 90.000,E1 331.897} C_DIS
LIN {X 0.040,Y -201.282,Z 1533.821,A 0.000,B 0.000,C 90.000,E1 327.788} C_DIS
LIN {X 0.077,Y -206.705,Z 1533.803,A 0.000,B 0.000,C 90.000,E1 324.562} C_DIS
LIN {X -0.023,Y -212.950,Z 1533.786,A 0.000,B 0.000,C 90.000,E1 321.412} C_DIS
LIN {X 0.108,Y -220.013,Z 1533.768,A 0.000,B 0.000,C 90.000,E1 318.243} C_DIS
LIN {X 0.025,Y -228.866,Z 1533.749,A 0.000,B 0.000,C 90.000,E1 314.798} C_DIS
LIN {X 0.096,Y -237.723,Z 1533.732,A 0.000,B 0.000,C 90.000,E1 311.757} C_DIS
LIN {X -0.050,Y -244.065,Z 1533.722,A 0.000,B 0.000,C 90.000,E1 309.930} C_DIS
LIN {X -0.063,Y -251.235,Z 1533.712,A 0.000,B 0.000,C 90.000,E1 308.096} C_DIS
LIN {X -0.149,Y -257.645,Z 1533.703,A 0.000,B 0.000,C 90.000,E1 306.664} C_DIS
LIN {X 0.061,Y -264.818,Z 1533.696,A 0.000,B 0.000,C 90.000,E1 305.185} C_DIS
LIN {X 0.066,Y -274.797,Z 1533.686,A 0.000,B 0.000,C 90.000,E1 303.420} C_DIS
LIN {X -0.076,Y -285.841,Z 1533.676,A 0.000,B 0.000,C 90.000,E1 301.720} C_DIS
LIN {X 0.053,Y -302.720,Z 1533.663,A 0.000,B 0.000,C 90.000,E1 299.333} C_DIS
LIN {X -0.067,Y -323.476,Z 1533.649,A 0.000,B 0.000,C 90.000,E1 296.744} C_DIS
LIN {X 0.153,Y -342.234,Z 1533.636,A 0.000,B 0.000,C 90.000,E1 294.515} C_DIS
LIN {X -0.030,Y -360.791,Z 1533.625,A 0.000,B 0.000,C 90.000,E1 292.514} C_DIS
LIN {X 0.079,Y -373.890,Z 1533.617,A 0.000,B 0.000,C 90.000,E1 291.099} C_DIS
LIN {X -0.036,Y -384.280,Z 1533.611,A 0.000,B 0.000,C 90.000,E1 289.993} C_DIS
LIN {X 0.066,Y -391.681,Z 1533.606,A 0.000,B 0.000,C 90.000,E1 289.141} C_DIS
LIN {X -0.068,Y -398.770,Z 1533.602,A 0.000,B 0.000,C 90.000,E1 288.308} C_DIS
LIN {X -0.018,Y -405.202,Z 1533.597,A 0.000,B 0.000,C 90.000,E1 287.457} C_DIS
LIN {X -0.025,Y -410.944,Z 1533.592,A 0.000,B 0.000,C 90.000,E1 286.622} C_DIS
LIN {X 0.018,Y -415.976,Z 1533.588,A 0.000,B 0.000,C 90.000,E1 285.788} C_DIS
LIN {X -0.024,Y -418.899,Z 1533.585,A 0.000,B 0.000,C 90.000,E1 285.245} C_DIS
LIN {X -0.011,Y -422.623,Z 1533.580,A 0.000,B 0.000,C 90.000,E1 284.426} C_DIS
LIN {X 0.140,Y -425.552,Z 1533.576,A 0.000,B 0.000,C 90.000,E1 283.592} C_DIS
LIN {X 0.045,Y -427.143,Z 1533.573,A 0.000,B 0.000,C 90.000,E1 283.063} C_DIS
LIN {X -0.039,Y -428.235,Z 1533.570,A 0.000,B 0.000,C 90.000,E1 282.535} C_DIS
LIN {X -0.113,Y -428.928,Z 1533.567,A 0.000,B 0.000,C 90.000,E1 282.007} C_DIS
LIN {X -0.180,Y -429.160,Z 1533.564,A 0.000,B 0.000,C 90.000,E1 281.478} C_DIS
LIN {X 0.175,Y -428.860,Z 1533.561,A 0.000,B 0.000,C 90.000,E1 280.894} C_DIS
LIN {X 0.109,Y -428.040,Z 1533.558,A 0.000,B 0.000,C 90.000,E1 280.366} C_DIS
LIN {X -0.033,Y -426.635,Z 1533.555,A 0.000,B 0.000,C 90.000,E1 279.849} C_DIS
LIN {X -0.107,Y -424.569,Z 1533.552,A 0.000,B 0.000,C 90.000,E1 279.321} C_DIS
LIN {X 0.161,Y -421.763,Z 1533.549,A 0.000,B 0.000,C 90.000,E1 278.746} C_DIS
LIN {X 0.055,Y -418.070,Z 1533.546,A 0.000,B 0.000,C 90.000,E1 278.219} C_DIS
LIN {X -0.129,Y -413.477,Z 1533.543,A 0.000,B 0.000,C 90.000,E1 277.701} C_DIS
LIN {X 0.075,Y -407.817,Z 1533.540,A 0.000,B 0.000,C 90.000,E1 277.125} C_DIS
LIN {X -0.154,Y -401.901,Z 1533.537,A 0.000,B 0.000,C 90.000,E1 276.663} C_DIS
LIN {X -0.063,Y -395.724,Z 1533.534,A 0.000,B 0.000,C 90.000,E1 276.201} C_DIS
LIN {X -0.055,Y -389.376,Z 1533.532,A 0.000,B 0.000,C 90.000,E1 275.796} C_DIS
LIN {X -0.150,Y -382.914,Z 1533.530,A 0.000,B 0.000,C 90.000,E1 275.448} C_DIS
LIN {X 0.114,Y -373.227,Z 1533.527,A 0.000,B 0.000,C 90.000,E1 274.935} C_DIS
LIN {X 0.121,Y -357.345,Z 1533.524,A 0.000,B 0.000,C 90.000,E1 274.245} C_DIS
LIN {X 0.117,Y -344.574,Z 1533.521,A 0.000,B 0.000,C 90.000,E1 273.726} C_DIS
LIN {X 0.068,Y -334.580,Z 1533.519,A 0.000,B 0.000,C 90.000,E1 273.383} C_DIS
LIN {X 0.040,Y -321.599,Z 1533.517,A 0.000,B 0.000,C 90.000,E1 272.980} C_DIS
LIN {X 0.072,Y -311.097,Z 1533.515,A 0.000,B 0.000,C 90.000,E1 272.694} C_DIS
LIN {X 0.069,Y -300.030,Z 1533.514,A 0.000,B 0.000,C 90.000,E1 272.465} C_DIS
LIN {X -0.044,Y -287.610,Z 1533.513,A 0.000,B 0.000,C 90.000,E1 272.293} C_DIS
LIN {X -0.124,Y -274.964,Z 1533.512,A 0.000,B 0.000,C 90.000,E1 272.178} C_DIS
LIN {X -0.069,Y -262.763,Z 1533.512,A 0.000,B 0.000,C 90.000,E1 272.121} C_DIS
LIN {X -0.066,Y -181.246,Z 1533.512,A 0.000,B 0.000,C 90.000,E1 272.121} C_DIS
LIN {X 0.016,Y -181.569,Z 1533.500,A 0.000,B 0.000,C 90.000,E1 270.057} C_DIS
LIN {X 0.004,Y -180.864,Z 1533.472,A 0.000,B 0.000,C 90.000,E1 265.008} C_DIS
LIN {X 0.058,Y -178.977,Z 1533.444,A 0.000,B 0.000,C 90.000,E1 259.926} C_DIS
LIN {X 0.068,Y -177.944,Z 1533.435,A 0.000,B 0.000,C 90.000,E1 258.229} C_DIS
LIN {X 0.082,Y -175.585,Z 1533.411,A 0.000,B 0.000,C 90.000,E1 253.976} C_DIS
LIN {X -0.074,Y -172.310,Z 1533.387,A 0.000,B 0.000,C 90.000,E1 249.752} C_DIS
LIN {X -0.094,Y -171.789,Z 1533.383,A 0.000,B 0.000,C 90.000,E1 248.901} C_DIS
LIN {X -0.057,Y -169.456,Z 1533.368,A 0.000,B 0.000,C 90.000,E1 246.305} C_DIS
LIN {X -0.001,Y -166.786,Z 1533.349,A 0.000,B 0.000,C 90.000,E1 242.820} C_DIS
LIN {X -0.005,Y -162.766,Z 1533.325,A 0.000,B 0.000,C 90.000,E1 238.456} C_DIS
LIN {X -0.030,Y -161.456,Z 1533.315,A 0.000,B 0.000,C 90.000,E1 236.707} C_DIS
LIN {X 0.012,Y -157.450,Z 1533.290,A 0.000,B 0.000,C 90.000,E1 232.271} C_DIS
LIN {X -0.055,Y -155.459,Z 1533.276,A 0.000,B 0.000,C 90.000,E1 229.622} C_DIS
LIN {X -0.013,Y -151.774,Z 1533.251,A 0.000,B 0.000,C 90.000,E1 225.121} C_DIS
LIN {X 0.003,Y -149.979,Z 1533.236,A 0.000,B 0.000,C 90.000,E1 222.405} C_DIS
LIN {X 0.015,Y -146.814,Z 1533.210,A 0.000,B 0.000,C 90.000,E1 217.855} C_DIS
LIN {X 0.031,Y -145.392,Z 1533.195,A 0.000,B 0.000,C 90.000,E1 215.105} C_DIS
LIN {X -0.051,Y -142.828,Z 1533.170,A 0.000,B 0.000,C 90.000,E1 210.541} C_DIS
LIN {X 0.005,Y -141.441,Z 1533.149,A 0.000,B 0.000,C 90.000,E1 206.821} C_DIS
LIN {X 0.050,Y -139.369,Z 1533.113,A 0.000,B 0.000,C 90.000,E1 200.301} C_DIS
LIN {X 0.036,Y -138.816,Z 1533.097,A 0.000,B 0.000,C 90.000,E1 197.511} C_DIS
LIN {X -0.049,Y -138.352,Z 1533.056,A 0.000,B 0.000,C 90.000,E1 190.074} C_DIS
LIN {X 0.063,Y -139.537,Z 1533.004,A 0.000,B 0.000,C 90.000,E1 180.688} C_DIS
LIN {X 0.016,Y -141.227,Z 1532.973,A 0.000,B 0.000,C 90.000,E1 175.122} C_DIS
LIN {X -0.025,Y -142.600,Z 1532.958,A 0.000,B 0.000,C 90.000,E1 172.356} C_DIS
LIN {X 0.069,Y -144.905,Z 1532.932,A 0.000,B 0.000,C 90.000,E1 167.701} C_DIS
LIN {X 0.022,Y -147.533,Z 1532.911,A 0.000,B 0.000,C 90.000,E1 164.047} C_DIS
LIN {X -0.046,Y -150.132,Z 1532.891,A 0.000,B 0.000,C 90.000,E1 160.423} C_DIS
LIN {X -0.035,Y -153.497,Z 1532.871,A 0.000,B 0.000,C 90.000,E1 156.794} C_DIS
LIN {X 0.028,Y -157.862,Z 1532.846,A 0.000,B 0.000,C 90.000,E1 152.281} C_DIS
LIN {X -0.016,Y -162.147,Z 1532.826,A 0.000,B 0.000,C 90.000,E1 148.742} C_DIS
LIN {X -0.037,Y -166.353,Z 1532.807,A 0.000,B 0.000,C 90.000,E1 145.229} C_DIS
LIN {X -0.031,Y -171.370,Z 1532.787,A 0.000,B 0.000,C 90.000,E1 141.743} C_DIS
LIN {X -0.106,Y -176.277,Z 1532.768,A 0.000,B 0.000,C 90.000,E1 138.324} C_DIS
LIN {X 0.012,Y -180.562,Z 1532.754,A 0.000,B 0.000,C 90.000,E1 135.729} C_DIS
LIN {X -0.009,Y -185.964,Z 1532.735,A 0.000,B 0.000,C 90.000,E1 132.366} C_DIS
LIN {X 0.047,Y -190.596,Z 1532.721,A 0.000,B 0.000,C 90.000,E1 129.850} C_DIS
LIN {X -0.046,Y -196.346,Z 1532.703,A 0.000,B 0.000,C 90.000,E1 126.583} C_DIS
LIN {X 0.032,Y -201.140,Z 1532.690,A 0.000,B 0.000,C 90.000,E1 124.119} C_DIS
LIN {X -0.034,Y -202.745,Z 1532.684,A 0.000,B 0.000,C 90.000,E1 123.214} C_DIS
LIN {X 0.161,Y -318.118,Z 1532.684,A 0.000,B 0.000,C 90.000,E1 123.166} C_DIS
LIN {X -0.077,Y -323.056,Z 1532.683,A 0.000,B 0.000,C 90.000,E1 123.038} C_DIS
LIN {X -0.144,Y -325.474,Z 1532.682,A 0.000,B 0.000,C 90.000,E1 122.880} C_DIS
LIN {X -0.181,Y -328.730,Z 1532.681,A 0.000,B 0.000,C 90.000,E1 122.546} C_DIS
LIN {X 0.089,Y -330.699,Z 1532.679,A 0.000,B 0.000,C 90.000,E1 122.212} C_DIS
LIN {X 0.080,Y -332.243,Z 1532.677,A 0.000,B 0.000,C 90.000,E1 121.926} C_DIS
LIN {X 0.120,Y -337.170,Z 1532.671,A 0.000,B 0.000,C 90.000,E1 120.669} C_DIS
LIN {X 0.103,Y -348.847,Z 1532.655,A 0.000,B 0.000,C 90.000,E1 117.897} C_DIS
LIN {X -0.089,Y -361.960,Z 1532.640,A 0.000,B 0.000,C 90.000,E1 115.207} C_DIS
LIN {X 0.120,Y -376.615,Z 1532.625,A 0.000,B 0.000,C 90.000,E1 112.514} C_DIS
LIN {X -0.188,Y -391.041,Z 1532.612,A 0.000,B 0.000,C 90.000,E1 110.248} C_DIS
LIN {X 0.104,Y -406.889,Z 1532.600,A 0.000,B 0.000,C 90.000,E1 107.946} C_DIS
LIN {X -0.240,Y -424.268,Z 1532.588,A 0.000,B 0.000,C 90.000,E1 105.788} C_DIS
LIN {X 0.146,Y -443.278,Z 1532.576,A 0.000,B 0.000,C 90.000,E1 103.592} C_DIS
LIN {X 0.056,Y -463.303,Z 1532.564,A 0.000,B 0.000,C 90.000,E1 101.591} C_DIS
LIN {X 0.221,Y -486.489,Z 1532.553,A 0.000,B 0.000,C 90.000,E1 99.500} C_DIS
LIN {X -0.026,Y -491.681,Z 1532.551,A 0.000,B 0.000,C 90.000,E1 99.095} C_DIS
LIN {X 0.125,Y -493.752,Z 1532.549,A 0.000,B 0.000,C 90.000,E1 98.859} C_DIS
LIN {X -0.213,Y -495.331,Z 1532.548,A 0.000,B 0.000,C 90.000,E1 98.681} C_DIS
LIN {X 0.117,Y -496.684,Z 1532.547,A 0.000,B 0.000,C 90.000,E1 98.398} C_DIS
LIN {X 0.029,Y -497.680,Z 1532.545,A 0.000,B 0.000,C 90.000,E1 98.163} C_DIS
LIN {X -0.201,Y -498.790,Z 1532.543,A 0.000,B 0.000,C 90.000,E1 97.701} C_DIS
LIN {X 0.069,Y -498.877,Z 1532.540,A 0.000,B 0.000,C 90.000,E1 97.182} C_DIS
LIN {X -0.148,Y -497.957,Z 1532.537,A 0.000,B 0.000,C 90.000,E1 96.720} C_DIS
LIN {X 0.130,Y -495.869,Z 1532.535,A 0.000,B 0.000,C 90.000,E1 96.201} C_DIS
LIN {X -0.069,Y -481.571,Z 1532.522,A 0.000,B 0.000,C 90.000,E1 94.012} C_DIS
LIN {X 0.051,Y -473.791,Z 1532.515,A 0.000,B 0.000,C 90.000,E1 92.751} C_DIS
LIN {X -0.145,Y -463.794,Z 1532.507,A 0.000,B 0.000,C 90.000,E1 91.260} C_DIS
LIN {X 0.167,Y -455.089,Z 1532.500,A 0.000,B 0.000,C 90.000,E1 89.943} C_DIS
LIN {X 0.098,Y -444.193,Z 1532.491,A 0.000,B 0.000,C 90.000,E1 88.396} C_DIS
LIN {X -0.124,Y -432.965,Z 1532.482,A 0.000,B 0.000,C 90.000,E1 86.846} C_DIS
LIN {X -0.126,Y -421.651,Z 1532.474,A 0.000,B 0.000,C 90.000,E1 85.241} C_DIS
LIN {X -0.141,Y -408.536,Z 1532.463,A 0.000,B 0.000,C 90.000,E1 83.337} C_DIS
LIN {X 0.118,Y -392.002,Z 1532.449,A 0.000,B 0.000,C 90.000,E1 80.792} C_DIS
LIN {X 0.086,Y -373.012,Z 1532.431,A 0.000,B 0.000,C 90.000,E1 77.645} C_DIS
LIN {X 0.114,Y -358.232,Z 1532.417,A 0.000,B 0.000,C 90.000,E1 74.991} C_DIS
LIN {X 0.020,Y -345.391,Z 1532.403,A 0.000,B 0.000,C 90.000,E1 72.598} C_DIS
LIN {X 0.044,Y -332.755,Z 1532.390,A 0.000,B 0.000,C 90.000,E1 70.134} C_DIS
LIN {X 0.105,Y -317.764,Z 1532.372,A 0.000,B 0.000,C 90.000,E1 66.975} C_DIS
LIN {X -0.028,Y -303.515,Z 1532.354,A 0.000,B 0.000,C 90.000,E1 63.768} C_DIS
LIN {X 0.090,Y -293.703,Z 1532.341,A 0.000,B 0.000,C 90.000,E1 61.435} C_DIS
LIN {X 0.068,Y -281.387,Z 1532.325,A 0.000,B 0.000,C 90.000,E1 58.408} C_DIS
LIN {X -0.029,Y -270.643,Z 1532.309,A 0.000,B 0.000,C 90.000,E1 55.674} C_DIS
LIN {X 0.013,Y -257.725,Z 1532.290,A 0.000,B 0.000,C 90.000,E1 52.145} C_DIS
LIN {X -0.119,Y -246.757,Z 1532.272,A 0.000,B 0.000,C 90.000,E1 48.933} C_DIS
LIN {X -0.039,Y -237.698,Z 1532.255,A 0.000,B 0.000,C 90.000,E1 45.972} C_DIS
LIN {X -0.009,Y -229.432,Z 1532.239,A 0.000,B 0.000,C 90.000,E1 42.975} C_DIS
LIN {X 0.011,Y -221.895,Z 1532.222,A 0.000,B 0.000,C 90.000,E1 39.930} C_DIS
LIN {X -0.089,Y -215.135,Z 1532.205,A 0.000,B 0.000,C 90.000,E1 36.870} C_DIS
LIN {X 0.034,Y -209.109,Z 1532.187,A 0.000,B 0.000,C 90.000,E1 33.706} C_DIS
LIN {X 0.002,Y -202.592,Z 1532.165,A 0.000,B 0.000,C 90.000,E1 29.745} C_DIS
LIN {X 0.005,Y -197.026,Z 1532.143,A 0.000,B 0.000,C 90.000,E1 25.720} C_DIS
LIN {X -0.051,Y -192.229,Z 1532.120,A 0.000,B 0.000,C 90.000,E1 21.663} C_DIS
LIN {X 0.069,Y -188.254,Z 1532.097,A 0.000,B 0.000,C 90.000,E1 17.511} C_DIS
LIN {X 0.040,Y -184.440,Z 1532.070,A 0.000,B 0.000,C 90.000,E1 12.535} C_DIS
LIN {X 0.056,Y -181.219,Z 1532.037,A 0.000,B 0.000,C 90.000,E1 6.663} C_DIS
LIN {X 0.056,Y -179.318,Z 1531.988,A 0.000,B 0.000,C 90.000,E1 357.822} C_DIS
LIN {X -0.031,Y -180.355,Z 1531.950,A 0.000,B 0.000,C 90.000,E1 351.084} C_DIS
LIN {X 0.010,Y -183.019,Z 1531.918,A 0.000,B 0.000,C 90.000,E1 345.172} C_DIS
LIN {X 0.055,Y -186.621,Z 1531.890,A 0.000,B 0.000,C 90.000,E1 340.134} C_DIS
LIN {X 0.005,Y -190.588,Z 1531.867,A 0.000,B 0.000,C 90.000,E1 335.997} C_DIS
LIN {X -0.044,Y -195.550,Z 1531.844,A 0.000,B 0.000,C 90.000,E1 331.897} C_DIS
LIN {X 0.102,Y -201.453,Z 1531.821,A 0.000,B 0.000,C 90.000,E1 327.788} C_DIS
LIN {X -0.025,Y -206.865,Z 1531.803,A 0.000,B 0.000,C 90.000,E1 324.609} C_DIS
LIN {X 0.050,Y -213.089,Z 1531.786,A 0.000,B 0.000,C 90.000,E1 321.412} C_DIS
LIN {X -0.124,Y -220.118,Z 1531.768,A 0.000,B 0.000,C 90.000,E1 318.324} C_DIS
LIN {X -0.051,Y -228.955,Z 1531.749,A 0.000,B 0.000,C 90.000,E1 314.838} C_DIS
LIN {X -0.149,Y -237.798,Z 1531.732,A 0.000,B 0.000,C 90.000,E1 311.838} C_DIS
LIN {X 0.045,Y -244.133,Z 1531.722,A 0.000,B 0.000,C 90.000,E1 309.930} C_DIS
LIN {X 0.034,Y -251.247,Z 1531.712,A 0.000,B 0.000,C 90.000,E1 308.096} C_DIS
LIN {X -0.048,Y -257.616,Z 1531.704,A 0.000,B 0.000,C 90.000,E1 306.664} C_DIS
LIN {X -0.053,Y -264.762,Z 1531.696,A 0.000,B 0.000,C 90.000,E1 305.231} C_DIS
LIN {X 0.021,Y -274.683,Z 1531.686,A 0.000,B 0.000,C 90.000,E1 303.452} C_DIS
LIN {X 0.032,Y -285.653,Z 1531.676,A 0.000,B 0.000,C 90.000,E1 301.720} C_DIS
LIN {X 0.032,Y -305.024,Z 1531.661,A 0.000,B 0.000,C 90.000,E1 299.027} C_DIS
LIN {X -0.016,Y -325.988,Z 1531.647,A 0.000,B 0.000,C 90.000,E1 296.437} C_DIS
LIN {X 0.043,Y -344.762,Z 1531.635,A 0.000,B 0.000,C 90.000,E1 294.259} C_DIS
LIN {X 0.078,Y -360.809,Z 1531.625,A 0.000,B 0.000,C 90.000,E1 292.514} C_DIS
LIN {X -0.040,Y -373.791,Z 1531.617,A 0.000,B 0.000,C 90.000,E1 291.153} C_DIS
LIN {X 0.218,Y -384.193,Z 1531.611,A 0.000,B 0.000,C 90.000,E1 289.993} C_DIS
LIN {X -0.188,Y -391.623,Z 1531.607,A 0.000,B 0.000,C 90.000,E1 289.214} C_DIS
LIN {X -0.198,Y -398.756,Z 1531.602,A 0.000,B 0.000,C 90.000,E1 288.362} C_DIS
LIN {X -0.153,Y -405.225,Z 1531.597,A 0.000,B 0.000,C 90.000,E1 287.511} C_DIS
LIN {X -0.163,Y -411.024,Z 1531.593,A 0.000,B 0.000,C 90.000,E1 286.677} C_DIS
LIN {X -0.124,Y -416.093,Z 1531.588,A 0.000,B 0.000,C 90.000,E1 285.843} C_DIS
LIN {X 0.238,Y -419.082,Z 1531.585,A 0.000,B 0.000,C 90.000,E1 285.245} C_DIS
LIN {X -0.155,Y -422.856,Z 1531.580,A 0.000,B 0.000,C 90.000,E1 284.481} C_DIS
LIN {X -0.005,Y -425.876,Z 1531.576,A 0.000,B 0.000,C 90.000,E1 283.647} C_DIS
LIN {X -0.099,Y -427.454,Z 1531.573,A 0.000,B 0.000,C 90.000,E1 283.119} C_DIS
LIN {X -0.181,Y -428.646,Z 1531.570,A 0.000,B 0.000,C 90.000,E1 282.591} C_DIS
LIN {X 0.165,Y -429.373,Z 1531.567,A 0.000,B 0.000,C 90.000,E1 282.007} C_DIS
LIN {X 0.099,Y -429.639,Z 1531.564,A 0.000,B 0.000,C 90.000,E1 281.478} C_DIS
LIN {X 0.035,Y -429.408,Z 1531.561,A 0.000,B 0.000,C 90.000,E1 280.950} C_DIS
LIN {X -0.027,Y -428.648,Z 1531.558,A 0.000,B 0.000,C 90.000,E1 280.423} C_DIS
LIN {X -0.168,Y -427.315,Z 1531.555,A 0.000,B 0.000,C 90.000,E1 279.905} C_DIS
LIN {X 0.181,Y -425.318,Z 1531.552,A 0.000,B 0.000,C 90.000,E1 279.321} C_DIS
LIN {X 0.034,Y -422.602,Z 1531.549,A 0.000,B 0.000,C 90.000,E1 278.803} C_DIS
LIN {X 0.193,Y -420.934,Z 1531.547,A 0.000,B 0.000,C 90.000,E1 278.511} C_DIS
LIN {X 0.021,Y -416.923,Z 1531.544,A 0.000,B 0.000,C 90.000,E1 277.992} C_DIS
LIN {X -0.112,Y -411.928,Z 1531.541,A 0.000,B 0.000,C 90.000,E1 277.466} C_DIS
LIN {X -0.119,Y -406.165,Z 1531.538,A 0.000,B 0.000,C 90.000,E1 276.947} C_DIS
LIN {X 0.186,Y -400.125,Z 1531.536,A 0.000,B 0.000,C 90.000,E1 276.429} C_DIS
LIN {X -0.064,Y -393.836,Z 1531.533,A 0.000,B 0.000,C 90.000,E1 276.030} C_DIS
LIN {X 0.043,Y -387.393,Z 1531.531,A 0.000,B 0.000,C 90.000,E1 275.625} C_DIS
LIN {X 0.114,Y -377.535,Z 1531.528,A 0.000,B 0.000,C 90.000,E1 275.106} C_DIS
LIN {X -0.100,Y -367.791,Z 1531.526,A 0.000,B 0.000,C 90.000,E1 274.702} C_DIS
LIN {X 0.047,Y -352.015,Z 1531.522,A 0.000,B 0.000,C 90.000,E1 274.012} C_DIS
LIN {X -0.165,Y -342.337,Z 1531.520,A 0.000,B 0.000,C 90.000,E1 273.669} C_DIS
LIN {X -0.168,Y -332.213,Z 1531.518,A 0.000,B 0.000,C 90.000,E1 273.326} C_DIS
LIN {X -0.133,Y -319.112,Z 1531.516,A 0.000,B 0.000,C 90.000,E1 272.922} C_DIS
LIN {X 0.001,Y -308.570,Z 1531.515,A 0.000,B 0.000,C 90.000,E1 272.636} C_DIS
LIN {X 0.066,Y -297.249,Z 1531.513,A 0.000,B 0.000,C 90.000,E1 272.407} C_DIS
LIN {X 0.016,Y -284.722,Z 1531.512,A 0.000,B 0.000,C 90.000,E1 272.236} C_DIS
LIN {X -0.080,Y -276.937,Z 1531.512,A 0.000,B 0.000,C 90.000,E1 272.178} C_DIS
LIN {X -0.063,Y -261.815,Z 1531.512,A 0.000,B 0.000,C 90.000,E1 272.121} C_DIS
LIN {X -0.064,Y -181.246,Z 1531.512,A 0.000,B 0.000,C 90.000,E1 272.121} C_DIS
LIN {X 0.033,Y -181.570,Z 1531.500,A 0.000,B 0.000,C 90.000,E1 270.057} C_DIS
LIN {X 0.022,Y -180.865,Z 1531.472,A 0.000,B 0.000,C 90.000,E1 265.008} C_DIS
LIN {X 0.074,Y -178.980,Z 1531.444,A 0.000,B 0.000,C 90.000,E1 259.926} C_DIS
LIN {X 0.084,Y -177.948,Z 1531.435,A 0.000,B 0.000,C 90.000,E1 258.229} C_DIS
LIN {X 0.099,Y -175.589,Z 1531.411,A 0.000,B 0.000,C 90.000,E1 253.976} C_DIS
LIN {X -0.057,Y -172.314,Z 1531.387,A 0.000,B 0.000,C 90.000,E1 249.752} C_DIS
LIN {X -0.078,Y -171.792,Z 1531.383,A 0.000,B 0.000,C 90.000,E1 248.901} C_DIS
LIN {X -0.040,Y -169.461,Z 1531.368,A 0.000,B 0.000,C 90.000,E1 246.305} C_DIS
LIN {X 0.016,Y -166.790,Z 1531.349,A 0.000,B 0.000,C 90.000,E1 242.820} C_DIS
LIN {X 0.011,Y -162.771,Z 1531.325,A 0.000,B 0.000,C 90.000,E1 238.456} C_DIS
LIN {X -0.014,Y -161.460,Z 1531.315,A 0.000,B 0.000,C 90.000,E1 236.707} C_DIS
LIN {X 0.028,Y -157.454,Z 1531.290,A 0.000,B 0.000,C 90.000,E1 232.271} C_DIS
LIN {X -0.038,Y -155.465,Z 1531.276,A 0.000,B 0.000,C 90.000,E1 229.622} C_DIS
LIN {X 0.002,Y -151.778,Z 1531.251,A 0.000,B 0.000,C 90.000,E1 225.121} C_DIS
LIN {X 0.019,Y -149.984,Z 1531.236,A 0.000,B 0.000,C 90.000,E1 222.405} C_DIS
LIN {X -0.060,Y -146.817,Z 1531.210,A 0.000,B 0.000,C 90.000,E1 217.890} C_DIS
LIN {X 0.046,Y -145.397,Z 1531.195,A 0.000,B 0.000,C 90.000,E1 215.105} C_DIS
LIN {X -0.037,Y -142.831,Z 1531.170,A 0.000,B 0.000,C 90.000,E1 210.541} C_DIS
LIN {X 0.020,Y -141.444,Z 1531.149,A 0.000,B 0.000,C 90.000,E1 206.821} C_DIS
LIN {X 0.065,Y -139.369,Z 1531.113,A 0.000,B 0.000,C 90.000,E1 200.301} C_DIS
LIN {X 0.050,Y -138.817,Z 1531.097,A 0.000,B 0.000,C 90.000,E1 197.511} C_DIS
LIN {X -0.035,Y -138.352,Z 1531.056,A 0.000,B 0.000,C 90.000,E1 190.074} C_DIS
LIN {X -0.062,Y -139.536,Z 1531.004,A 0.000,B 0.000,C 90.000,E1 180.745} C_DIS
LIN {X 0.031,Y -141.225,Z 1530.973,A 0.000,B 0.000,C 90.000,E1 175.122} C_DIS
LIN {X -0.011,Y -142.597,Z 1530.958,A 0.000,B 0.000,C 90.000,E1 172.356} C_DIS
LIN {X -0.057,Y -144.902,Z 1530.932,A 0.000,B 0.000,C 90.000,E1 167.757} C_DIS
LIN {X 0.037,Y -147.530,Z 1530.911,A 0.000,B 0.000,C 90.000,E1 164.047} C_DIS
LIN {X -0.031,Y -150.128,Z 1530.891,A 0.000,B 0.000,C 90.000,E1 160.423} C_DIS
LIN {X -0.019,Y -153.491,Z 1530.871,A 0.000,B 0.000,C 90.000,E1 156.794} C_DIS
LIN {X 0.044,Y -157.855,Z 1530.846,A 0.000,B 0.000,C 90.000,E1 152.281} C_DIS
LIN {X 0.000,Y -162.140,Z 1530.826,A 0.000,B 0.000,C 90.000,E1 148.742} C_DIS
LIN {X -0.021,Y -166.346,Z 1530.807,A 0.000,B 0.000,C 90.000,E1 145.229} C_DIS
LIN {X -0.016,Y -171.362,Z 1530.787,A 0.000,B 0.000,C 90.000,E1 141.743} C_DIS
LIN {X -0.089,Y -176.268,Z 1530.768,A 0.000,B 0.000,C 90.000,E1 138.324} C_DIS
LIN {X 0.030,Y -180.552,Z 1530.754,A 0.000,B 0.000,C 90.000,E1 135.729} C_DIS
LIN {X 0.009,Y -185.954,Z 1530.735,A 0.000,B 0.000,C 90.000,E1 132.366} C_DIS
LIN {X 0.065,Y -190.586,Z 1530.721,A 0.000,B 0.000,C 90.000,E1 129.850} C_DIS
LIN {X -0.027,Y -196.336,Z 1530.703,A 0.000,B 0.000,C 90.000,E1 126.583} C_DIS
LIN {X 0.050,Y -201.132,Z 1530.690,A 0.000,B 0.000,C 90.000,E1 124.119} C_DIS
LIN {X -0.008,Y -202.676,Z 1530.685,A 0.000,B 0.000,C 90.000,E1 123.245} C_DIS
LIN {X -0.047,Y -316.938,Z 1530.685,A 0.000,B 0.000,C 90.000,E1 123.245} C_DIS
LIN {X -0.076,Y -319.500,Z 1530.684,A 0.000,B 0.000,C 90.000,E1 123.214} C_DIS
LIN {X -0.047,Y -323.388,Z 1530.683,A 0.000,B 0.000,C 90.000,E1 123.038} C_DIS
LIN {X -0.114,Y -325.664,Z 1530.682,A 0.000,B 0.000,C 90.000,E1 122.880} C_DIS
LIN {X -0.151,Y -328.804,Z 1530.681,A 0.000,B 0.000,C 90.000,E1 122.546} C_DIS
LIN {X 0.075,Y -330.767,Z 1530.679,A 0.000,B 0.000,C 90.000,E1 122.212} C_DIS
LIN {X 0.022,Y -332.302,Z 1530.677,A 0.000,B 0.000,C 90.000,E1 121.926} C_DIS
LIN {X -0.130,Y -347.505,Z 1530.657,A 0.000,B 0.000,C 90.000,E1 118.231} C_DIS
LIN {X 0.124,Y -360.455,Z 1530.642,A 0.000,B 0.000,C 90.000,E1 115.463} C_DIS
LIN {X -0.050,Y -374.940,Z 1530.627,A 0.000,B 0.000,C 90.000,E1 112.823} C_DIS
LIN {X 0.094,Y -389.203,Z 1530.614,A 0.000,B 0.000,C 90.000,E1 110.482} C_DIS
LIN {X -0.042,Y -404.874,Z 1530.601,A 0.000,B 0.000,C 90.000,E1 108.236} C_DIS
LIN {X -0.043,Y -422.062,Z 1530.589,A 0.000,B 0.000,C 90.000,E1 106.024} C_DIS
LIN {X -0.151,Y -440.887,Z 1530.577,A 0.000,B 0.000,C 90.000,E1 103.883} C_DIS
LIN {X 0.028,Y -460.842,Z 1530.566,A 0.000,B 0.000,C 90.000,E1 101.827} C_DIS
LIN {X 0.117,Y -483.933,Z 1530.554,A 0.000,B 0.000,C 90.000,E1 99.726} C_DIS
LIN {X -0.092,Y -491.727,Z 1530.550,A 0.000,B 0.000,C 90.000,E1 99.095} C_DIS
LIN {X 0.052,Y -493.771,Z 1530.549,A 0.000,B 0.000,C 90.000,E1 98.859} C_DIS
LIN {X 0.194,Y -495.330,Z 1530.548,A 0.000,B 0.000,C 90.000,E1 98.624} C_DIS
LIN {X 0.035,Y -496.659,Z 1530.547,A 0.000,B 0.000,C 90.000,E1 98.398} C_DIS
LIN {X -0.052,Y -497.635,Z 1530.545,A 0.000,B 0.000,C 90.000,E1 98.163} C_DIS
LIN {X 0.210,Y -498.713,Z 1530.543,A 0.000,B 0.000,C 90.000,E1 97.644} C_DIS
LIN {X -0.013,Y -498.771,Z 1530.540,A 0.000,B 0.000,C 90.000,E1 97.182} C_DIS
LIN {X -0.231,Y -497.819,Z 1530.537,A 0.000,B 0.000,C 90.000,E1 96.720} C_DIS
LIN {X 0.046,Y -495.692,Z 1530.534,A 0.000,B 0.000,C 90.000,E1 96.201} C_DIS
LIN {X -0.023,Y -482.907,Z 1530.524,A 0.000,B 0.000,C 90.000,E1 94.245} C_DIS
LIN {X 0.142,Y -475.189,Z 1530.517,A 0.000,B 0.000,C 90.000,E1 92.980} C_DIS
LIN {X 0.166,Y -466.999,Z 1530.510,A 0.000,B 0.000,C 90.000,E1 91.718} C_DIS
LIN {X 0.060,Y -458.433,Z 1530.503,A 0.000,B 0.000,C 90.000,E1 90.458} C_DIS
LIN {X -0.156,Y -449.498,Z 1530.495,A 0.000,B 0.000,C 90.000,E1 89.198} C_DIS
LIN {X 0.139,Y -438.474,Z 1530.487,A 0.000,B 0.000,C 90.000,E1 87.593} C_DIS
LIN {X -0.039,Y -425.315,Z 1530.476,A 0.000,B 0.000,C 90.000,E1 85.755} C_DIS
LIN {X 0.056,Y -410.332,Z 1530.464,A 0.000,B 0.000,C 90.000,E1 83.571} C_DIS
LIN {X -0.036,Y -393.771,Z 1530.450,A 0.000,B 0.000,C 90.000,E1 81.084} C_DIS
LIN {X -0.027,Y -376.315,Z 1530.435,A 0.000,B 0.000,C 90.000,E1 78.229} C_DIS
LIN {X 0.009,Y -361.433,Z 1530.420,A 0.000,B 0.000,C 90.000,E1 75.589} C_DIS
LIN {X -0.038,Y -350.159,Z 1530.408,A 0.000,B 0.000,C 90.000,E1 73.504} C_DIS
LIN {X 0.103,Y -337.429,Z 1530.395,A 0.000,B 0.000,C 90.000,E1 71.040} C_DIS
LIN {X 0.013,Y -320.669,Z 1530.376,A 0.000,B 0.000,C 90.000,E1 67.614} C_DIS
LIN {X -0.038,Y -306.238,Z 1530.358,A 0.000,B 0.000,C 90.000,E1 64.409} C_DIS
LIN {X 0.124,Y -297.844,Z 1530.347,A 0.000,B 0.000,C 90.000,E1 62.410} C_DIS
LIN {X 0.096,Y -286.771,Z 1530.332,A 0.000,B 0.000,C 90.000,E1 59.744} C_DIS
LIN {X 0.032,Y -277.353,Z 1530.319,A 0.000,B 0.000,C 90.000,E1 57.375} C_DIS
LIN {X -0.005,Y -266.721,Z 1530.303,A 0.000,B 0.000,C 90.000,E1 54.609} C_DIS
LIN {X -0.003,Y -256.551,Z 1530.288,A 0.000,B 0.000,C 90.000,E1 51.778} C_DIS
LIN {X -0.008,Y -245.690,Z 1530.270,A 0.000,B 0.000,C 90.000,E1 48.528} C_DIS
LIN {X 0.017,Y -235.694,Z 1530.251,A 0.000,B 0.000,C 90.000,E1 45.202} C_DIS
LIN {X 0.005,Y -227.634,Z 1530.234,A 0.000,B 0.000,C 90.000,E1 42.204} C_DIS
LIN {X 0.011,Y -220.337,Z 1530.218,A 0.000,B 0.000,C 90.000,E1 39.152} C_DIS
LIN {X -0.120,Y -213.808,Z 1530.200,A 0.000,B 0.000,C 90.000,E1 36.091} C_DIS
LIN {X 0.028,Y -207.972,Z 1530.183,A 0.000,B 0.000,C 90.000,E1 32.911} C_DIS
LIN {X -0.032,Y -201.691,Z 1530.161,A 0.000,B 0.000,C 90.000,E1 28.949} C_DIS
LIN {X 0.027,Y -196.285,Z 1530.138,A 0.000,B 0.000,C 90.000,E1 24.899} C_DIS
LIN {X -0.055,Y -191.620,Z 1530.116,A 0.000,B 0.000,C 90.000,E1 20.844} C_DIS
LIN {X 0.097,Y -187.809,Z 1530.093,A 0.000,B 0.000,C 90.000,E1 16.677} C_DIS
LIN {X 0.054,Y -184.690,Z 1530.070,A 0.000,B 0.000,C 90.000,E1 12.535} C_DIS
LIN {X 0.081,Y -181.474,Z 1530.037,A 0.000,B 0.000,C 90.000,E1 6.663} C_DIS
LIN {X 0.059,Y -179.591,Z 1529.988,A 0.000,B 0.000,C 90.000,E1 357.822} C_DIS
LIN {X 0.056,Y -180.879,Z 1529.946,A 0.000,B 0.000,C 90.000,E1 350.218} C_DIS
LIN {X 0.020,Y -183.772,Z 1529.913,A 0.000,B 0.000,C 90.000,E1 344.338} C_DIS
LIN {X -0.022,Y -187.578,Z 1529.885,A 0.000,B 0.000,C 90.000,E1 339.337} C_DIS
LIN {X 0.031,Y -191.713,Z 1529.862,A 0.000,B 0.000,C 90.000,E1 335.177} C_DIS
LIN {X 0.109,Y -196.811,Z 1529.839,A 0.000,B 0.000,C 90.000,E1 331.051} C_DIS
LIN {X -0.048,Y -202.904,Z 1529.817,A 0.000,B 0.000,C 90.000,E1 327.041} C_DIS
LIN {X -0.023,Y -208.480,Z 1529.799,A 0.000,B 0.000,C 90.000,E1 323.829} C_DIS
LIN {X 0.058,Y -214.891,Z 1529.781,A 0.000,B 0.000,C 90.000,E1 320.642} C_DIS
LIN {X -0.066,Y -222.094,Z 1529.764,A 0.000,B 0.000,C 90.000,E1 317.553} C_DIS
LIN {X -0.098,Y -231.149,Z 1529.745,A 0.000,B 0.000,C 90.000,E1 314.109} C_DIS
LIN {X 0.060,Y -239.092,Z 1529.730,A 0.000,B 0.000,C 90.000,E1 311.434} C_DIS
LIN {X 0.124,Y -245.574,Z 1529.720,A 0.000,B 0.000,C 90.000,E1 309.564} C_DIS
LIN {X 0.135,Y -252.808,Z 1529.710,A 0.000,B 0.000,C 90.000,E1 307.729} C_DIS
LIN {X 0.074,Y -259.318,Z 1529.702,A 0.000,B 0.000,C 90.000,E1 306.297} C_DIS
LIN {X -0.003,Y -268.539,Z 1529.692,A 0.000,B 0.000,C 90.000,E1 304.532} C_DIS
LIN {X 0.136,Y -278.816,Z 1529.682,A 0.000,B 0.000,C 90.000,E1 302.752} C_DIS
LIN {X 0.034,Y -292.545,Z 1529.671,A 0.000,B 0.000,C 90.000,E1 300.718} C_DIS
LIN {X 0.120,Y -315.152,Z 1529.654,A 0.000,B 0.000,C 90.000,E1 297.719} C_DIS
LIN {X 0.058,Y -333.566,Z 1529.642,A 0.000,B 0.000,C 90.000,E1 295.540} C_DIS
LIN {X 0.076,Y -352.135,Z 1529.630,A 0.000,B 0.000,C 90.000,E1 293.462} C_DIS
LIN {X 0.003,Y -368.174,Z 1529.621,A 0.000,B 0.000,C 90.000,E1 291.770} C_DIS
LIN {X -0.011,Y -381.244,Z 1529.613,A 0.000,B 0.000,C 90.000,E1 290.375} C_DIS
LIN {X 0.080,Y -388.835,Z 1529.609,A 0.000,B 0.000,C 90.000,E1 289.523} C_DIS
LIN {X 0.127,Y -396.094,Z 1529.604,A 0.000,B 0.000,C 90.000,E1 288.671} C_DIS
LIN {X 0.163,Y -402.867,Z 1529.599,A 0.000,B 0.000,C 90.000,E1 287.819} C_DIS
LIN {X 0.131,Y -408.974,Z 1529.594,A 0.000,B 0.000,C 90.000,E1 286.985} C_DIS
LIN {X -0.235,Y -414.375,Z 1529.590,A 0.000,B 0.000,C 90.000,E1 286.205} C_DIS
LIN {X -0.163,Y -419.064,Z 1529.585,A 0.000,B 0.000,C 90.000,E1 285.371} C_DIS
LIN {X -0.041,Y -422.929,Z 1529.581,A 0.000,B 0.000,C 90.000,E1 284.537} C_DIS
LIN {X 0.008,Y -426.037,Z 1529.576,A 0.000,B 0.000,C 90.000,E1 283.716} C_DIS
LIN {X 0.014,Y -427.680,Z 1529.573,A 0.000,B 0.000,C 90.000,E1 283.175} C_DIS
LIN {X -0.067,Y -428.935,Z 1529.570,A 0.000,B 0.000,C 90.000,E1 282.647} C_DIS
LIN {X -0.140,Y -429.754,Z 1529.567,A 0.000,B 0.000,C 90.000,E1 282.119} C_DIS
LIN {X 0.215,Y -430.098,Z 1529.564,A 0.000,B 0.000,C 90.000,E1 281.535} C_DIS
LIN {X 0.153,Y -429.972,Z 1529.561,A 0.000,B 0.000,C 90.000,E1 281.007} C_DIS
LIN {X 0.013,Y -429.303,Z 1529.558,A 0.000,B 0.000,C 90.000,E1 280.489} C_DIS
LIN {X -0.047,Y -428.069,Z 1529.555,A 0.000,B 0.000,C 90.000,E1 279.962} C_DIS
LIN {X -0.114,Y -426.200,Z 1529.552,A 0.000,B 0.000,C 90.000,E1 279.434} C_DIS
LIN {X 0.161,Y -423.633,Z 1529.549,A 0.000,B 0.000,C 90.000,E1 278.859} C_DIS
LIN {X 0.003,Y -420.221,Z 1529.546,A 0.000,B 0.000,C 90.000,E1 278.341} C_DIS
LIN {X -0.110,Y -415.863,Z 1529.543,A 0.000,B 0.000,C 90.000,E1 277.814} C_DIS
LIN {X 0.106,Y -410.555,Z 1529.540,A 0.000,B 0.000,C 90.000,E1 277.239} C_DIS
LIN {X 0.131,Y -404.552,Z 1529.537,A 0.000,B 0.000,C 90.000,E1 276.720} C_DIS
LIN {X 0.160,Y -398.458,Z 1529.535,A 0.000,B 0.000,C 90.000,E1 276.258} C_DIS
LIN {X 0.077,Y -392.092,Z 1529.533,A 0.000,B 0.000,C 90.000,E1 275.853} C_DIS
LIN {X -0.134,Y -385.515,Z 1529.531,A 0.000,B 0.000,C 90.000,E1 275.511} C_DIS
LIN {X -0.017,Y -379.013,Z 1529.529,A 0.000,B 0.000,C 90.000,E1 275.163} C_DIS
LIN {X -0.013,Y -366.115,Z 1529.526,A 0.000,B 0.000,C 90.000,E1 274.588} C_DIS
LIN {X -0.095,Y -350.568,Z 1529.522,A 0.000,B 0.000,C 90.000,E1 273.955} C_DIS
LIN {X 0.030,Y -340.661,Z 1529.520,A 0.000,B 0.000,C 90.000,E1 273.555} C_DIS
LIN {X 0.092,Y -330.683,Z 1529.518,A 0.000,B 0.000,C 90.000,E1 273.212} C_DIS
LIN {X 0.143,Y -317.404,Z 1529.516,A 0.000,B 0.000,C 90.000,E1 272.808} C_DIS
LIN {X -0.014,Y -306.275,Z 1529.514,A 0.000,B 0.000,C 90.000,E1 272.579} C_DIS
LIN {X 0.111,Y -294.812,Z 1529.513,A 0.000,B 0.000,C 90.000,E1 272.350} C_DIS
LIN {X 0.111,Y -281.913,Z 1529.512,A 0.000,B 0.000,C 90.000,E1 272.178} C_DIS
LIN {X 0.032,Y -269.079,Z 1529.512,A 0.000,B 0.000,C 90.000,E1 272.121} C_DIS
LIN {X -0.033,Y -263.007,Z 1529.512,A 0.000,B 0.000,C 90.000,E1 272.121} C_DIS
LIN {X -0.045,Y -181.245,Z 1529.512,A 0.000,B 0.000,C 90.000,E1 272.121} C_DIS
LIN {X 0.070,Y -181.571,Z 1529.500,A 0.000,B 0.000,C 90.000,E1 270.057} C_DIS
LIN {X 0.058,Y -180.868,Z 1529.472,A 0.000,B 0.000,C 90.000,E1 265.008} C_DIS
LIN {X -0.065,Y -178.982,Z 1529.444,A 0.000,B 0.000,C 90.000,E1 259.982} C_DIS
LIN {X -0.054,Y -177.955,Z 1529.435,A 0.000,B 0.000,C 90.000,E1 258.285} C_DIS
LIN {X -0.034,Y -175.598,Z 1529.411,A 0.000,B 0.000,C 90.000,E1 254.031} C_DIS
LIN {X -0.021,Y -172.322,Z 1529.387,A 0.000,B 0.000,C 90.000,E1 249.752} C_DIS
LIN {X -0.043,Y -171.799,Z 1529.383,A 0.000,B 0.000,C 90.000,E1 248.901} C_DIS
LIN {X -0.005,Y -169.472,Z 1529.368,A 0.000,B 0.000,C 90.000,E1 246.305} C_DIS
LIN {X 0.051,Y -166.799,Z 1529.349,A 0.000,B 0.000,C 90.000,E1 242.820} C_DIS
LIN {X 0.045,Y -162.781,Z 1529.325,A 0.000,B 0.000,C 90.000,E1 238.456} C_DIS
LIN {X 0.020,Y -161.469,Z 1529.315,A 0.000,B 0.000,C 90.000,E1 236.707} C_DIS
LIN {X 0.062,Y -157.464,Z 1529.291,A 0.000,B 0.000,C 90.000,E1 232.271} C_DIS
LIN {X -0.006,Y -155.477,Z 1529.276,A 0.000,B 0.000,C 90.000,E1 229.622} C_DIS
LIN {X -0.072,Y -151.787,Z 1529.251,A 0.000,B 0.000,C 90.000,E1 225.162} C_DIS
LIN {X -0.059,Y -149.995,Z 1529.236,A 0.000,B 0.000,C 90.000,E1 222.447} C_DIS
LIN {X -0.028,Y -146.825,Z 1529.210,A 0.000,B 0.000,C 90.000,E1 217.890} C_DIS
LIN {X -0.041,Y -145.405,Z 1529.195,A 0.000,B 0.000,C 90.000,E1 215.152} C_DIS
LIN {X -0.005,Y -142.836,Z 1529.170,A 0.000,B 0.000,C 90.000,E1 210.541} C_DIS
LIN {X -0.074,Y -141.450,Z 1529.149,A 0.000,B 0.000,C 90.000,E1 206.873} C_DIS
LIN {X -0.034,Y -139.371,Z 1529.113,A 0.000,B 0.000,C 90.000,E1 200.355} C_DIS
LIN {X 0.040,Y -138.820,Z 1529.097,A 0.000,B 0.000,C 90.000,E1 197.528} C_DIS
LIN {X -0.003,Y -138.353,Z 1529.056,A 0.000,B 0.000,C 90.000,E1 190.074} C_DIS
LIN {X -0.031,Y -139.534,Z 1529.004,A 0.000,B 0.000,C 90.000,E1 180.745} C_DIS
LIN {X 0.062,Y -141.219,Z 1528.973,A 0.000,B 0.000,C 90.000,E1 175.122} C_DIS
LIN {X 0.021,Y -142.592,Z 1528.958,A 0.000,B 0.000,C 90.000,E1 172.356} C_DIS
LIN {X -0.025,Y -144.894,Z 1528.932,A 0.000,B 0.000,C 90.000,E1 167.757} C_DIS
LIN {X -0.071,Y -147.521,Z 1528.911,A 0.000,B 0.000,C 90.000,E1 164.102} C_DIS
LIN {X 0.003,Y -150.117,Z 1528.891,A 0.000,B 0.000,C 90.000,E1 160.423} C_DIS
LIN {X 0.014,Y -153.478,Z 1528.871,A 0.000,B 0.000,C 90.000,E1 156.794} C_DIS
LIN {X 0.077,Y -157.841,Z 1528.846,A 0.000,B 0.000,C 90.000,E1 152.281} C_DIS
LIN {X 0.034,Y -162.126,Z 1528.826,A 0.000,B 0.000,C 90.000,E1 148.742} C_DIS
LIN {X 0.014,Y -166.330,Z 1528.807,A 0.000,B 0.000,C 90.000,E1 145.229} C_DIS
LIN {X 0.020,Y -171.347,Z 1528.787,A 0.000,B 0.000,C 90.000,E1 141.743} C_DIS
LIN {X -0.052,Y -176.251,Z 1528.768,A 0.000,B 0.000,C 90.000,E1 138.324} C_DIS
LIN {X 0.067,Y -180.531,Z 1528.754,A 0.000,B 0.000,C 90.000,E1 135.729} C_DIS
LIN {X 0.046,Y -185.934,Z 1528.735,A 0.000,B 0.000,C 90.000,E1 132.366} C_DIS
LIN {X -0.019,Y -190.565,Z 1528.722,A 0.000,B 0.000,C 90.000,E1 129.886} C_DIS
LIN {X 0.011,Y -196.315,Z 1528.703,A 0.000,B 0.000,C 90.000,E1 126.583} C_DIS
LIN {X 0.089,Y -201.113,Z 1528.690,A 0.000,B 0.000,C 90.000,E1 124.119} C_DIS
LIN {X -0.070,Y -202.622,Z 1528.685,A 0.000,B 0.000,C 90.000,E1 123.293} C_DIS
LIN {X -0.145,Y -317.414,Z 1528.685,A 0.000,B 0.000,C 90.000,E1 123.293} C_DIS
LIN {X -0.014,Y -320.130,Z 1528.684,A 0.000,B 0.000,C 90.000,E1 123.214} C_DIS
LIN {X -0.051,Y -325.770,Z 1528.683,A 0.000,B 0.000,C 90.000,E1 122.880} C_DIS
LIN {X -0.088,Y -328.828,Z 1528.681,A 0.000,B 0.000,C 90.000,E1 122.546} C_DIS
LIN {X 0.106,Y -330.784,Z 1528.679,A 0.000,B 0.000,C 90.000,E1 122.212} C_DIS
LIN {X 0.019,Y -332.310,Z 1528.677,A 0.000,B 0.000,C 90.000,E1 121.926} C_DIS
LIN {X 0.173,Y -346.134,Z 1528.658,A 0.000,B 0.000,C 90.000,E1 118.487} C_DIS
LIN {X -0.086,Y -358.925,Z 1528.643,A 0.000,B 0.000,C 90.000,E1 115.796} C_DIS
LIN {X 0.194,Y -373.230,Z 1528.628,A 0.000,B 0.000,C 90.000,E1 113.078} C_DIS
LIN {X -0.053,Y -387.323,Z 1528.615,A 0.000,B 0.000,C 90.000,E1 110.791} C_DIS
LIN {X 0.144,Y -402.812,Z 1528.603,A 0.000,B 0.000,C 90.000,E1 108.489} C_DIS
LIN {X -0.176,Y -419.804,Z 1528.590,A 0.000,B 0.000,C 90.000,E1 106.315} C_DIS
LIN {X 0.075,Y -438.416,Z 1528.578,A 0.000,B 0.000,C 90.000,E1 104.120} C_DIS
LIN {X 0.101,Y -458.284,Z 1528.567,A 0.000,B 0.000,C 90.000,E1 102.063} C_DIS
LIN {X -0.087,Y -478.725,Z 1528.557,A 0.000,B 0.000,C 90.000,E1 100.197} C_DIS
LIN {X -0.102,Y -491.701,Z 1528.550,A 0.000,B 0.000,C 90.000,E1 99.095} C_DIS
LIN {X 0.037,Y -493.731,Z 1528.549,A 0.000,B 0.000,C 90.000,E1 98.859} C_DIS
LIN {X 0.176,Y -495.280,Z 1528.548,A 0.000,B 0.000,C 90.000,E1 98.624} C_DIS
LIN {X 0.016,Y -496.599,Z 1528.547,A 0.000,B 0.000,C 90.000,E1 98.398} C_DIS
LIN {X -0.071,Y -497.566,Z 1528.545,A 0.000,B 0.000,C 90.000,E1 98.163} C_DIS
LIN {X 0.192,Y -498.627,Z 1528.543,A 0.000,B 0.000,C 90.000,E1 97.644} C_DIS
LIN {X -0.033,Y -498.670,Z 1528.540,A 0.000,B 0.000,C 90.000,E1 97.182} C_DIS
LIN {X -0.251,Y -497.704,Z 1528.537,A 0.000,B 0.000,C 90.000,E1 96.720} C_DIS
LIN {X 0.026,Y -495.559,Z 1528.534,A 0.000,B 0.000,C 90.000,E1 96.201} C_DIS
LIN {X -0.047,Y -482.763,Z 1528.524,A 0.000,B 0.000,C 90.000,E1 94.245} C_DIS
LIN {X -0.060,Y -473.475,Z 1528.515,A 0.000,B 0.000,C 90.000,E1 92.751} C_DIS
LIN {X 0.204,Y -463.511,Z 1528.507,A 0.000,B 0.000,C 90.000,E1 91.203} C_DIS
